KUKA KRL program: MyProgram_166().src

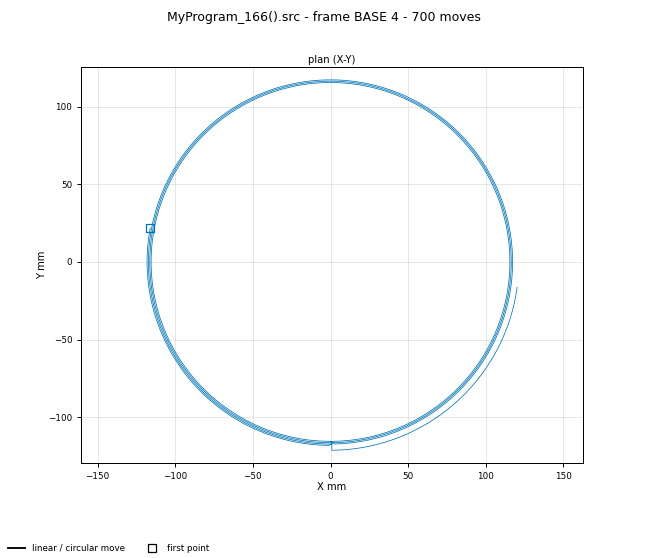
[picture p0: tool path of MyProgram_166().src in frame BASE 4, 700 of 700 moves have a stored position in this frame; points joined in program order, loops and branches not executed]
&ACCESS RVP
&REL 1
&PARAM TEMPLATE = C:\KRC\Roboter\Template\vorgabe
&PARAM EDITMASK = *
DEF MyProgram_166()
; ---- Setting reference (Base) ----
$BASE = BASE_DATA[4]

; --------------------------
; ---- Setting tool (TCP) ----
$TOOL = TOOL_DATA[3]
; --------------------------

$VEL.CP = VEL_APROX_PRINT
Startdeposition()
$VEL.CP = VEL_PRINT
LIN {X -116.0779,Y 21.7482,Z 125,A 166.5415,B 24.9441,C -1.7272,E1 24.8419,E2 279.4054} C_DIS
LIN {X -116.9015,Y 16.7566,Z 125,A 168.4487,B 24.9461,C -1.6962,E1 24.8412,E2 277.5607} C_DIS
LIN {X -117.4117,Y 12.7035,Z 125,A 170.2727,B 24.9469,C -1.6831,E1 24.8406,E2 275.757} C_DIS
LIN {X -117.7284,Y 9.3134,Z 125,A 171.8723,B 24.9474,C -1.6755,E1 24.8402,E2 274.1658} C_DIS
LIN {X -118.0302,Y 3.9618,Z 125,A 174.4618,B 24.948,C -1.6666,E1 24.8399,E2 271.5821} C_DIS
LIN {X -118.095,Y 0.6382,Z 125,A 176.1945,B 24.948,C -1.6663,E1 24.8398,E2 269.8396} C_DIS
LIN {X -118.0463,Y -3.4397,Z 125,A 178.1568,B 24.9484,C -1.6592,E1 24.8398,E2 267.8824} C_DIS
LIN {X -117.9024,Y -6.7675,Z 125,A 179.7767,B 24.9487,C -1.6541,E1 24.8401,E2 266.265} C_DIS
LIN {X -117.4382,Y -12.4501,Z 125,A -177.4787,B 24.9493,C -1.6442,E1 24.8408,E2 263.5274} C_DIS
LIN {X -117.0347,Y -15.812,Z 125,A -175.2833,B 24.9482,C -1.6622,E1 24.8416,E2 261.2762} C_DIS
LIN {X -116.456,Y -19.6147,Z 125,A -173.0042,B 24.9475,C -1.6738,E1 24.8427,E2 258.9558} C_DIS
LIN {X -115.3606,Y -25.2717,Z 125,A -171.1064,B 24.9504,C -1.627,E1 24.8438,E2 257.1584} C_DIS
LIN {X -113.6862,Y -31.9722,Z 125,A -167.6075,B 24.9507,C -1.6228,E1 24.8462,E2 253.6492} C_DIS
LIN {X -112.4267,Y -36.1525,Z 125,A -165.5854,B 24.9513,C -1.6123,E1 24.8479,E2 251.6404} C_DIS
LIN {X -111.457,Y -39.0393,Z 125,A -164.0611,B 24.9514,C -1.6098,E1 24.8493,E2 250.1133} C_DIS
LIN {X -110.0528,Y -42.8395,Z 125,A -162.0909,B 24.9518,C -1.6041,E1 24.8512,E2 248.1455} C_DIS
LIN {X -108.7242,Y -46.1068,Z 125,A -159.2633,B 24.9492,C -1.6468,E1 24.8545,E2 245.2007} C_DIS
LIN {X -105.8827,Y -52.303,Z 125,A -157.3666,B 24.9534,C -1.5771,E1 24.8566,E2 243.4597} C_DIS
LIN {X -103.1276,Y -57.545,Z 125,A -154.1935,B 24.9531,C -1.5818,E1 24.8608,E2 240.2585} C_DIS
LIN {X -101.6073,Y -60.1887,Z 125,A -152.6604,B 24.9532,C -1.5801,E1 24.8629,E2 238.7217} C_DIS
LIN {X -97.5843,Y -66.5143,Z 125,A -149.0981,B 24.954,C -1.5673,E1 24.8683,E2 235.1718} C_DIS
LIN {X -95.9307,Y -68.8777,Z 125,A -147.6463,B 24.954,C -1.566,E1 24.8706,E2 233.716} C_DIS
LIN {X -93.6134,Y -71.9949,Z 125,A -145.7524,B 24.9543,C -1.5617,E1 24.8738,E2 231.8231} C_DIS
LIN {X -91.4931,Y -74.6719,Z 125,A -144.0977,B 24.9545,C -1.5577,E1 24.8767,E2 230.1705} C_DIS
LIN {X -88.0813,Y -78.6665,Z 125,A -141.3029,B 24.9543,C -1.5623,E1 24.8819,E2 227.3518} C_DIS
LIN {X -85.8212,Y -81.1267,Z 125,A -139.7844,B 24.9547,C -1.5543,E1 24.8848,E2 225.8458} C_DIS
LIN {X -82.07,Y -84.9191,Z 125,A -137.0977,B 24.9548,C -1.553,E1 24.8901,E2 223.1508} C_DIS
LIN {X -78.6307,Y -88.1133,Z 125,A -134.9895,B 24.9555,C -1.5411,E1 24.8944,E2 221.0626} C_DIS
LIN {X -72.9131,Y -92.9008,Z 125,A -131.3391,B 24.9558,C -1.5355,E1 24.9023,E2 217.4116} C_DIS
LIN {X -68.4919,Y -96.206,Z 125,A -128.6806,B 24.9561,C -1.53,E1 24.9083,E2 214.7569} C_DIS
LIN {X -65.9216,Y -97.9856,Z 125,A -127.1661,B 24.9563,C -1.5274,E1 24.9117,E2 213.2434} C_DIS
LIN {X -62.3775,Y -100.2787,Z 125,A -125.0915,B 24.9564,C -1.5253,E1 24.9166,E2 211.167} C_DIS
LIN {X -58.5723,Y -102.548,Z 125,A -122.9855,B 24.9567,C -1.5203,E1 24.9217,E2 209.0667} C_DIS
LIN {X -55.7443,Y -104.1139,Z 125,A -120.7068,B 24.955,C -1.5497,E1 24.9275,E2 206.7118} C_DIS
LIN {X -51.6289,Y -106.2142,Z 125,A -119.1905,B 24.957,C -1.5146,E1 24.9311,E2 205.2748} C_DIS
LIN {X -48.5348,Y -107.6619,Z 125,A -117.4642,B 24.957,C -1.5158,E1 24.9355,E2 203.5415} C_DIS
LIN {X -42.3143,Y -110.2565,Z 125,A -114.3104,B 24.9574,C -1.5072,E1 24.9436,E2 200.401} C_DIS
LIN {X -39.7247,Y -111.2164,Z 125,A -112.6586,B 24.9567,C -1.5199,E1 24.948,E2 198.7157} C_DIS
LIN {X -35.4891,Y -112.6389,Z 125,A -110.3493,B 24.9565,C -1.5246,E1 24.9542,E2 196.3911} C_DIS
LIN {X -30.9043,Y -113.9809,Z 125,A -108.3462,B 24.9573,C -1.5089,E1 24.9595,E2 194.4221} C_DIS
LIN {X -27.7382,Y -114.7927,Z 125,A -106.8062,B 24.9575,C -1.5059,E1 24.9636,E2 192.8869} C_DIS
LIN {X -24.3093,Y -115.5686,Z 125,A -104.9791,B 24.9573,C -1.5106,E1 24.9687,E2 191.0466} C_DIS
LIN {X -20.8405,Y -116.2428,Z 125,A -103.3413,B 24.9575,C -1.5065,E1 24.9731,E2 189.4166} C_DIS
LIN {X -17.1768,Y -116.8418,Z 125,A -101.1085,B 24.9564,C -1.5257,E1 24.9794,E2 187.1365} C_DIS
LIN {X -13.728,Y -117.2956,Z 125,A -99.9123,B 24.9577,C -1.503,E1 24.9826,E2 185.9933} C_DIS
LIN {X -10.8458,Y -117.5971,Z 125,A -98.4243,B 24.9575,C -1.5066,E1 24.9868,E2 184.4959} C_DIS
LIN {X -7.1405,Y -117.8818,Z 125,A -96.3974,B 24.9569,C -1.5168,E1 24.9925,E2 182.444} C_DIS
LIN {X -1.2408,Y -118.0908,Z 125,A -93.9033,B 24.9578,C -1.5003,E1 24.9993,E2 179.9888} C_DIS
LIN {X -1.2408,Y -118.0908,Z 125,A -93.9033,B 24.9578,C -1.5003,E1 24.9993,E2 179.9888} C_DIS
Enddeposition()
LIN {X 0.8351,Y -117.2293,Z 125,A -92.7873,B 24.9567,C -1.5205,E1 25.0026,E2 178.825} C_DIS
Startdeposition()
$VEL.CP = VEL_PRINT
LIN {X -1.6148,Y -117.2225,Z 125,A -94.8526,B 24.9589,C -1.4811,E1 24.9966,E2 180.9837} C_DIS
LIN {X -6.2337,Y -117.0668,Z 125,A -96.9986,B 24.9586,C -1.4859,E1 24.9906,E2 183.1186} C_DIS
LIN {X -9.7696,Y -116.8254,Z 125,A -98.7217,B 24.9586,C -1.4863,E1 24.9858,E2 184.8415} C_DIS
LIN {X -13.4236,Y -116.4615,Z 125,A -100.2293,B 24.9579,C -1.4993,E1 24.9817,E2 186.3191} C_DIS
LIN {X -17.0983,Y -115.9804,Z 125,A -102.4267,B 24.9588,C -1.4825,E1 24.9755,E2 188.5581} C_DIS
LIN {X -20.6841,Y -115.3933,Z 125,A -104.0258,B 24.9584,C -1.4909,E1 24.9712,E2 190.1388} C_DIS
LIN {X -23.7178,Y -114.8082,Z 125,A -105.6383,B 24.9586,C -1.487,E1 24.9667,E2 191.7624} C_DIS
LIN {X -27.5658,Y -113.9457,Z 125,A -107.5616,B 24.9586,C -1.4882,E1 24.9615,E2 193.6855} C_DIS
LIN {X -31.5414,Y -112.9104,Z 125,A -109.9728,B 24.9594,C -1.4718,E1 24.9549,E2 196.1393} C_DIS
LIN {X -34.9646,Y -111.8972,Z 125,A -111.6053,B 24.9591,C -1.478,E1 24.9505,E2 197.7599} C_DIS
LIN {X -39.9943,Y -110.1995,Z 125,A -113.8892,B 24.9582,C -1.4937,E1 24.9446,E2 200.0108} C_DIS
LIN {X -42.7939,Y -109.1427,Z 125,A -115.7888,B 24.9592,C -1.4762,E1 24.9396,E2 201.9561} C_DIS
LIN {X -46.2472,Y -107.7268,Z 125,A -117.2748,B 24.9583,C -1.4927,E1 24.9358,E2 203.4063} C_DIS
LIN {X -49.5329,Y -106.2541,Z 125,A -118.8769,B 24.9578,C -1.5016,E1 24.9318,E2 204.9913} C_DIS
LIN {X -54.7369,Y -103.6693,Z 125,A -121.9132,B 24.958,C -1.4967,E1 24.9242,E2 208.0474} C_DIS
LIN {X -59.799,Y -100.8343,Z 125,A -124.7248,B 24.9577,C -1.5018,E1 24.9174,E2 210.8553} C_DIS
LIN {X -63.9365,Y -98.2653,Z 125,A -127.107,B 24.9575,C -1.5053,E1 24.9118,E2 213.2365} C_DIS
LIN {X -67.376,Y -95.9386,Z 125,A -129.3507,B 24.9579,C -1.4996,E1 24.9066,E2 215.5015} C_DIS
LIN {X -71.4168,Y -92.9683,Z 125,A -131.5025,B 24.9569,C -1.5167,E1 24.9018,E2 217.6203} C_DIS
LIN {X -73.3854,Y -91.4238,Z 125,A -133.2937,B 24.9581,C -1.4949,E1 24.8978,E2 219.47} C_DIS
LIN {X -76.5724,Y -88.7728,Z 125,A -134.9135,B 24.9569,C -1.516,E1 24.8945,E2 221.0461} C_DIS
LIN {X -79.2536,Y -86.3846,Z 125,A -136.6869,B 24.9568,C -1.5188,E1 24.8908,E2 222.8199} C_DIS
LIN {X -81.8829,Y -83.8994,Z 125,A -138.5802,B 24.9568,C -1.5172,E1 24.887,E2 224.7249} C_DIS
LIN {X -85.2057,Y -80.5202,Z 125,A -140.8343,B 24.9564,C -1.5249,E1 24.8826,E2 226.9703} C_DIS
LIN {X -88.1501,Y -77.2854,Z 125,A -142.9732,B 24.9562,C -1.5297,E1 24.8786,E2 229.1073} C_DIS
LIN {X -91.033,Y -73.8677,Z 125,A -144.9562,B 24.9554,C -1.5434,E1 24.8751,E2 231.0669} C_DIS
LIN {X -93.5183,Y -70.6958,Z 125,A -146.9961,B 24.9553,C -1.5452,E1 24.8716,E2 233.1121} C_DIS
LIN {X -95.4795,Y -68.0229,Z 125,A -148.6269,B 24.9551,C -1.5489,E1 24.869,E2 234.7422} C_DIS
LIN {X -97.7454,Y -64.7249,Z 125,A -151.0294,B 24.9558,C -1.5354,E1 24.8652,E2 237.1887} C_DIS
LIN {X -99.8083,Y -61.5001,Z 125,A -152.5944,B 24.9548,C -1.553,E1 24.8629,E2 238.7199} C_DIS
LIN {X -102.0444,Y -57.7129,Z 125,A -154.8515,B 24.9548,C -1.5544,E1 24.8598,E2 240.9854} C_DIS
LIN {X -104.1752,Y -53.7698,Z 125,A -156.8916,B 24.954,C -1.5667,E1 24.8571,E2 243.0071} C_DIS
LIN {X -106.0255,Y -50.024,Z 125,A -159.5909,B 24.9552,C -1.5456,E1 24.8538,E2 245.7713} C_DIS
LIN {X -107.9815,Y -45.6448,Z 125,A -161.2325,B 24.9532,C -1.5811,E1 24.8521,E2 247.3372} C_DIS
LIN {X -109.202,Y -42.6428,Z 125,A -162.8678,B 24.953,C -1.5837,E1 24.8504,E2 248.9757} C_DIS
LIN {X -110.5039,Y -39.1465,Z 125,A -164.7261,B 24.9528,C -1.5877,E1 24.8486,E2 250.8349} C_DIS
LIN {X -111.655,Y -35.7315,Z 125,A -166.5622,B 24.9526,C -1.5899,E1 24.847,E2 252.676} C_DIS
LIN {X -112.8242,Y -31.8458,Z 125,A -169.1513,B 24.9537,C -1.5714,E1 24.845,E2 255.3243} C_DIS
LIN {X -114.074,Y -27.037,Z 125,A -170.9059,B 24.9517,C -1.6063,E1 24.8439,E2 257.006} C_DIS
LIN {X -115.1522,Y -21.9871,Z 125,A -173.4355,B 24.9512,C -1.614,E1 24.8424,E2 259.5321} C_DIS
LIN {X -116.2866,Y -14.8631,Z 125,A -176.9173,B 24.9504,C -1.627,E1 24.841,E2 263.0037} C_DIS
LIN {X -116.6475,Y -11.7067,Z 125,A -178.8834,B 24.9511,C -1.6152,E1 24.8404,E2 265.0097} C_DIS
LIN {X -116.9276,Y -8.4665,Z 125,A 179.86,B 24.95,C -1.6339,E1 24.8401,E2 266.2295} C_DIS
LIN {X -117.1256,Y -5.0025,Z 125,A 178.1548,B 24.9497,C -1.639,E1 24.8399,E2 267.9326} C_DIS
LIN {X -117.2264,Y -1.3455,Z 125,A 176.2701,B 24.9495,C -1.6409,E1 24.8398,E2 269.8242} C_DIS
LIN {X -117.2105,Y 2.2703,Z 125,A 174.6527,B 24.9488,C -1.6527,E1 24.8398,E2 271.423} C_DIS
LIN {X -117.0681,Y 6.2092,Z 125,A 172.3947,B 24.9493,C -1.6456,E1 24.8401,E2 273.7118} C_DIS
LIN {X -116.7635,Y 10.4787,Z 125,A 170.5424,B 24.9482,C -1.6621,E1 24.8405,E2 275.5357} C_DIS
LIN {X -116.1042,Y 16.2268,Z 125,A 167.5686,B 24.948,C -1.6654,E1 24.8415,E2 278.5195} C_DIS
LIN {X -115.4155,Y 20.5602,Z 125,A 165.5301,B 24.9473,C -1.6767,E1 24.8425,E2 280.5433} C_DIS
LIN {X -114.1275,Y 26.8053,Z 125,A 162.2668,B 24.9471,C -1.6808,E1 24.8444,E2 283.816} C_DIS
LIN {X -112.9284,Y 31.478,Z 125,A 159.9483,B 24.9465,C -1.6899,E1 24.846,E2 286.1263} C_DIS
LIN {X -112.0005,Y 34.6314,Z 125,A 158.3319,B 24.9462,C -1.6946,E1 24.8474,E2 287.7407} C_DIS
LIN {X -110.8147,Y 38.2607,Z 125,A 156.4862,B 24.9458,C -1.7013,E1 24.849,E2 289.581} C_DIS
LIN {X -108.853,Y 43.5312,Z 125,A 153.6729,B 24.9454,C -1.7072,E1 24.8518,E2 292.396} C_DIS
LIN {X -107.4588,Y 46.8619,Z 125,A 151.9605,B 24.9449,C -1.7148,E1 24.8537,E2 294.0998} C_DIS
LIN {X -105.8573,Y 50.3772,Z 125,A 150.0068,B 24.9447,C -1.7179,E1 24.856,E2 296.0569} C_DIS
LIN {X -104.1375,Y 53.8435,Z 125,A 147.8473,B 24.945,C -1.7126,E1 24.8587,E2 298.2405} C_DIS
LIN {X -101.4971,Y 58.6675,Z 125,A 144.7651,B 24.9455,C -1.7046,E1 24.863,E2 301.3579} C_DIS
LIN {X -98.9869,Y 62.8124,Z 125,A 143.1773,B 24.9431,C -1.7431,E1 24.8653,E2 302.8621} C_DIS
LIN {X -95.8292,Y 67.5327,Z 125,A 139.7815,B 24.9442,C -1.7255,E1 24.8707,E2 306.3166} C_DIS
LIN {X -93.5753,Y 70.6199,Z 125,A 138.8928,B 24.9412,C -1.7708,E1 24.872,E2 307.1016} C_DIS
LIN {X -91.6258,Y 73.1332,Z 125,A 136.9431,B 24.942,C -1.7586,E1 24.8754,E2 309.0896} C_DIS
LIN {X -89.5071,Y 75.7106,Z 125,A 135.1595,B 24.9422,C -1.7566,E1 24.8786,E2 310.8862} C_DIS
LIN {X -87.2439,Y 78.3068,Z 125,A 133.6175,B 24.9415,C -1.7668,E1 24.8814,E2 312.4109} C_DIS
LIN {X -84.5415,Y 81.2171,Z 125,A 131.5821,B 24.9415,C -1.7678,E1 24.8853,E2 314.4529} C_DIS
LIN {X -81.1171,Y 84.6378,Z 125,A 129.058,B 24.9415,C -1.7669,E1 24.8904,E2 316.9895} C_DIS
LIN {X -77.8834,Y 87.623,Z 125,A 126.6566,B 24.9418,C -1.7616,E1 24.8954,E2 319.4132} C_DIS
LIN {X -75.3603,Y 89.803,Z 125,A 125.2726,B 24.9409,C -1.7754,E1 24.8983,E2 320.7697} C_DIS
LIN {X -72.6864,Y 91.979,Z 125,A 123.3436,B 24.9413,C -1.769,E1 24.9026,E2 322.721} C_DIS
LIN {X -70.1029,Y 93.9637,Z 125,A 121.5268,B 24.9417,C -1.7631,E1 24.9067,E2 324.5585} C_DIS
LIN {X -66.7194,Y 96.3951,Z 125,A 119.9213,B 24.9403,C -1.7851,E1 24.9103,E2 326.1172} C_DIS
LIN {X -64.0955,Y 98.1604,Z 125,A 118.303,B 24.9403,C -1.7851,E1 24.9141,E2 327.7408} C_DIS
LIN {X -61.2043,Y 99.988,Z 125,A 116.6727,B 24.94,C -1.7899,E1 24.9179,E2 329.3646} C_DIS
LIN {X -57.3374,Y 102.2541,Z 125,A 114.5912,B 24.9394,C -1.7984,E1 24.9229,E2 331.432} C_DIS
LIN {X -54.0312,Y 104.0408,Z 125,A 112.8232,B 24.939,C -1.8044,E1 24.9272,E2 333.1908} C_DIS
LIN {X -48.6263,Y 106.6732,Z 125,A 109.7819,B 24.939,C -1.8047,E1 24.9349,E2 336.2391} C_DIS
LIN {X -45.4531,Y 108.0623,Z 125,A 108.1017,B 24.9387,C -1.8078,E1 24.9392,E2 337.916} C_DIS
LIN {X -39.0031,Y 110.5542,Z 125,A 104.7495,B 24.9384,C -1.8134,E1 24.948,E2 341.2617} C_DIS
LIN {X -35.6874,Y 111.6693,Z 125,A 102.4145,B 24.94,C -1.7889,E1 24.9543,E2 343.6592} C_DIS
LIN {X -31.5151,Y 112.9171,Z 125,A 100.777,B 24.9385,C -1.812,E1 24.9586,E2 345.2443} C_DIS
LIN {X -23.9618,Y 114.7581,Z 125,A 97.0607,B 24.938,C -1.8192,E1 24.9687,E2 348.9488} C_DIS
LIN {X -20.7726,Y 115.3774,Z 125,A 95.4352,B 24.938,C -1.8188,E1 24.9731,E2 350.5768} C_DIS
LIN {X -16.7737,Y 116.0265,Z 125,A 93.482,B 24.9378,C -1.8213,E1 24.9785,E2 352.5258} C_DIS
LIN {X -13.0492,Y 116.5054,Z 125,A 91.5989,B 24.9378,C -1.8203,E1 24.9837,E2 354.4126} C_DIS
LIN {X -9.6564,Y 116.8344,Z 125,A 89.9798,B 24.9377,C -1.8232,E1 24.9882,E2 356.0256} C_DIS
LIN {X -6.466,Y 117.0539,Z 125,A 88.4343,B 24.9377,C -1.8245,E1 24.9925,E2 357.5684} C_DIS
LIN {X -2.5675,Y 117.205,Z 125,A 86.4811,B 24.9377,C -1.8231,E1 24.998,E2 359.5254} C_DIS
LIN {X 0.8052,Y 117.2297,Z 125,A 84.8525,B 24.9377,C -1.8243,E1 25.0025,E2 361.1511} C_DIS
LIN {X 4.8542,Y 117.132,Z 125,A 82.9127,B 24.9375,C -1.8262,E1 25.0079,E2 363.0858} C_DIS
LIN {X 8.3744,Y 116.9338,Z 125,A 81.1059,B 24.9377,C -1.8225,E1 25.013,E2 364.9007} C_DIS
LIN {X 11.9675,Y 116.6202,Z 125,A 79.4204,B 24.9375,C -1.8257,E1 25.0176,E2 366.5776} C_DIS
LIN {X 15.1732,Y 116.2464,Z 125,A 77.8138,B 24.9376,C -1.8241,E1 25.0221,E2 368.1868} C_DIS
LIN {X 18.973,Y 115.6875,Z 125,A 75.8997,B 24.9378,C -1.8219,E1 25.0274,E2 370.1043} C_DIS
LIN {X 22.6611,Y 115.0224,Z 125,A 74.0299,B 24.938,C -1.8194,E1 25.0325,E2 371.9778} C_DIS
LIN {X 26.259,Y 114.2537,Z 125,A 72.3871,B 24.9375,C -1.8254,E1 25.037,E2 373.6042} C_DIS
LIN {X 31.9221,Y 112.8025,Z 125,A 69.1138,B 24.9389,C -1.805,E1 25.0459,E2 376.9205} C_DIS
LIN {X 35.1622,Y 111.8359,Z 125,A 67.7111,B 24.9383,C -1.8149,E1 25.0496,E2 378.2975} C_DIS
LIN {X 39.4824,Y 110.386,Z 125,A 65.1137,B 24.9395,C -1.7963,E1 25.0565,E2 380.9335} C_DIS
LIN {X 43.0096,Y 109.0579,Z 125,A 63.7611,B 24.9382,C -1.8165,E1 25.0599,E2 382.2355} C_DIS
LIN {X 46.5591,Y 107.5908,Z 125,A 62.1231,B 24.9376,C -1.8252,E1 25.0641,E2 383.8489} C_DIS
LIN {X 50.5222,Y 105.7876,Z 125,A 59.5155,B 24.9392,C -1.801,E1 25.0708,E2 386.5072} C_DIS
LIN {X 55.0343,Y 103.5126,Z 125,A 57.2937,B 24.9387,C -1.8089,E1 25.0763,E2 388.704} C_DIS
LIN {X 58.1162,Y 101.8138,Z 125,A 55.5703,B 24.9388,C -1.8063,E1 25.0805,E2 390.4285} C_DIS
LIN {X 61.5238,Y 99.7934,Z 125,A 53.5557,B 24.9393,C -1.7998,E1 25.0853,E2 392.4523} C_DIS
LIN {X 64.3245,Y 98.0095,Z 125,A 51.3769,B 24.9412,C -1.7719,E1 25.0905,E2 394.6897} C_DIS
LIN {X 68.1982,Y 95.3544,Z 125,A 49.7395,B 24.9394,C -1.798,E1 25.0941,E2 396.26} C_DIS
LIN {X 73.4759,Y 91.3505,Z 125,A 46.4859,B 24.9399,C -1.7913,E1 25.1013,E2 399.5175} C_DIS
LIN {X 76.1243,Y 89.1546,Z 125,A 44.995,B 24.9395,C -1.7968,E1 25.1045,E2 400.9895} C_DIS
LIN {X 78.7411,Y 86.8548,Z 125,A 43.1919,B 24.94,C -1.7887,E1 25.1082,E2 402.8046} C_DIS
LIN {X 81.3986,Y 84.3665,Z 125,A 41.3875,B 24.9404,C -1.7838,E1 25.1119,E2 404.6131} C_DIS
LIN {X 84.8199,Y 80.9275,Z 125,A 39.072,B 24.9405,C -1.7812,E1 25.1164,E2 406.9249} C_DIS
LIN {X 87.4068,Y 78.1248,Z 125,A 37.2011,B 24.9408,C -1.7766,E1 25.12,E2 408.7982} C_DIS
LIN {X 89.8127,Y 75.3486,Z 125,A 35.5173,B 24.9408,C -1.7776,E1 25.123,E2 410.4721} C_DIS
LIN {X 93.0756,Y 71.2775,Z 125,A 32.7485,B 24.9419,C -1.7612,E1 25.1279,E2 413.2667} C_DIS
LIN {X 97.1409,Y 65.6284,Z 125,A 29.4447,B 24.9421,C -1.7571,E1 25.1332,E2 416.5641} C_DIS
LIN {X 99.395,Y 62.1617,Z 125,A 27.5293,B 24.9421,C -1.7567,E1 25.136,E2 418.4708} C_DIS
LIN {X 100.6871,Y 60.0479,Z 125,A 25.6319,B 24.9445,C -1.7213,E1 25.1389,E2 420.442} C_DIS
LIN {X 102.9107,Y 56.1507,Z 125,A 24.0908,B 24.9429,C -1.7458,E1 25.1409,E2 421.9173} C_DIS
LIN {X 104.2182,Y 53.6856,Z 125,A 22.891,B 24.9426,C -1.7497,E1 25.1424,E2 423.1015} C_DIS
LIN {X 105.5158,Y 51.0879,Z 125,A 21.253,B 24.9436,C -1.7353,E1 25.1444,E2 424.7647} C_DIS
LIN {X 106.9734,Y 47.9601,Z 125,A 19.6193,B 24.9437,C -1.733,E1 25.1463,E2 426.3951} C_DIS
LIN {X 108.5068,Y 44.3819,Z 125,A 17.8754,B 24.9436,C -1.7349,E1 25.1482,E2 428.1248} C_DIS
LIN {X 109.8782,Y 40.8741,Z 125,A 15.821,B 24.9446,C -1.7193,E1 25.1503,E2 430.2046} C_DIS
LIN {X 110.8838,Y 38.0607,Z 125,A 13.7234,B 24.9468,C -1.6848,E1 25.1523,E2 432.3716} C_DIS
LIN {X 112.3926,Y 33.3367,Z 125,A 11.4302,B 24.9468,C -1.6835,E1 25.154,E2 434.6548} C_DIS
LIN {X 113.5969,Y 28.9696,Z 125,A 9.8432,B 24.9454,C -1.7063,E1 25.1551,E2 436.179} C_DIS
LIN {X 114.5094,Y 25.1205,Z 125,A 7.9293,B 24.9458,C -1.7012,E1 25.1563,E2 438.0939} C_DIS
LIN {X 115.254,Y 21.4586,Z 125,A 5.9882,B 24.9465,C -1.6899,E1 25.1574,E2 440.0503} C_DIS
LIN {X 115.8309,Y 18.074,Z 125,A 4.4194,B 24.9465,C -1.6898,E1 25.1581,E2 441.6101} C_DIS
LIN {X 116.3583,Y 14.3051,Z 125,A 2.5225,B 24.947,C -1.682,E1 25.1588,E2 443.5142} C_DIS
LIN {X 116.7249,Y 10.8971,Z 125,A 0.9515,B 24.947,C -1.6816,E1 25.1592,E2 445.0768} C_DIS
LIN {X 116.9915,Y 7.5207,Z 125,A -0.808,B 24.9477,C -1.6712,E1 25.1595,E2 446.8502} C_DIS
LIN {X 117.1775,Y 3.5875,Z 125,A -2.6481,B 24.9477,C -1.669,E1 25.1597,E2 448.6846} C_DIS
LIN {X 117.2324,Y -0.4409,Z 125,A -4.6079,B 24.9482,C -1.663,E1 25.1597,E2 450.6469} C_DIS
LIN {X 117.1621,Y -4.0889,Z 125,A -6.2539,B 24.9482,C -1.6637,E1 25.1597,E2 452.2814} C_DIS
LIN {X 117.0279,Y -6.9364,Z 125,A -7.8163,B 24.9489,C -1.6511,E1 25.1594,E2 453.8644} C_DIS
LIN {X 116.7319,Y -10.821,Z 125,A -9.6054,B 24.9489,C -1.6504,E1 25.159,E2 455.6445} C_DIS
LIN {X 116.3079,Y -14.6987,Z 125,A -11.5635,B 24.9495,C -1.6416,E1 25.1584,E2 457.6116} C_DIS
LIN {X 115.7525,Y -18.5812,Z 125,A -13.4711,B 24.9499,C -1.6358,E1 25.1576,E2 459.5217} C_DIS
LIN {X 115.0246,Y -22.6497,Z 125,A -15.5647,B 24.9505,C -1.6257,E1 25.1565,E2 461.6268} C_DIS
LIN {X 114.0065,Y -27.3162,Z 125,A -17.5785,B 24.95,C -1.6335,E1 25.1553,E2 463.6106} C_DIS
LIN {X 112.2087,Y -33.9568,Z 125,A -21.0165,B 24.9509,C -1.619,E1 25.1527,E2 467.063} C_DIS
LIN {X 110.3917,Y -39.4659,Z 125,A -23.9646,B 24.9518,C -1.6046,E1 25.1501,E2 470.0284} C_DIS
LIN {X 109.0827,Y -42.9465,Z 125,A -25.693,B 24.9518,C -1.6032,E1 25.1483,E2 471.7506} C_DIS
LIN {X 107.9815,Y -45.6448,Z 125,A -27.637,B 24.9536,C -1.5741,E1 25.1462,E2 473.7525} C_DIS
LIN {X 106.33,Y -49.3697,Z 125,A -29.6176,B 24.9539,C -1.5685,E1 25.1438,E2 475.7356} C_DIS
LIN {X 104.5358,Y -53.0641,Z 125,A -30.9535,B 24.9524,C -1.5944,E1 25.1423,E2 477.0034} C_DIS
LIN {X 101.108,Y -59.3358,Z 125,A -34.5861,B 24.9534,C -1.5773,E1 25.1373,E2 480.6573} C_DIS
LIN {X 98.6083,Y -63.4023,Z 125,A -36.856,B 24.9536,C -1.5736,E1 25.1339,E2 482.9245} C_DIS
LIN {X 94.9914,Y -68.7062,Z 125,A -39.9233,B 24.9539,C -1.568,E1 25.1291,E2 485.9899} C_DIS
LIN {X 92.367,Y -72.1953,Z 125,A -42.2211,B 24.9547,C -1.5544,E1 25.1252,E2 488.3089} C_DIS
LIN {X 89.4516,Y -75.7757,Z 125,A -44.5234,B 24.9552,C -1.5462,E1 25.121,E2 490.6199} C_DIS
LIN {X 85.9649,Y -79.7104,Z 125,A -47.0053,B 24.9554,C -1.5437,E1 25.1164,E2 493.0966} C_DIS
LIN {X 82.9275,Y -82.8668,Z 125,A -49.6064,B 24.9569,C -1.5168,E1 25.1112,E2 495.7502} C_DIS
LIN {X 79.9206,Y -85.769,Z 125,A -51.0702,B 24.9556,C -1.539,E1 25.1083,E2 497.1555} C_DIS
LIN {X 77.0081,Y -88.3924,Z 125,A -53.0042,B 24.9559,C -1.5337,E1 25.1043,E2 499.0944} C_DIS
LIN {X 73.7199,Y -91.1528,Z 125,A -55.9662,B 24.9585,C -1.4888,E1 25.0977,E2 502.1512} C_DIS
LIN {X 69.1598,Y -94.6593,Z 125,A -58.4359,B 24.9579,C -1.4986,E1 25.0922,E2 504.589} C_DIS
LIN {X 65.6786,Y -97.1069,Z 125,A -59.9349,B 24.9566,C -1.5214,E1 25.0889,E2 506.0291} C_DIS
LIN {X 62.4525,Y -99.2133,Z 125,A -61.9006,B 24.9571,C -1.5138,E1 25.0842,E2 508.0063} C_DIS
LIN {X 58.2312,Y -101.7477,Z 125,A -64.8395,B 24.9587,C -1.4848,E1 25.077,E2 511.0049} C_DIS
LIN {X 54.2238,Y -103.9395,Z 125,A -66.4275,B 24.9572,C -1.5106,E1 25.0732,E2 512.5273} C_DIS
LIN {X 51.658,Y -105.2383,Z 125,A -68.2403,B 24.9584,C -1.4895,E1 25.0686,E2 514.3852} C_DIS
LIN {X 48.4985,Y -106.7308,Z 125,A -69.5497,B 24.9576,C -1.5051,E1 25.0654,E2 515.6542} C_DIS
LIN {X 45.4161,Y -108.0779,Z 125,A -71.2077,B 24.9577,C -1.502,E1 25.0611,E2 517.3157} C_DIS
LIN {X 41.49,Y -109.645,Z 125,A -73.4705,B 24.9584,C -1.4901,E1 25.0551,E2 519.6017} C_DIS
LIN {X 38.4727,Y -110.7403,Z 125,A -75.1612,B 24.9588,C -1.4825,E1 25.0507,E2 521.3071} C_DIS
LIN {X 35.2715,Y -111.802,Z 125,A -76.5266,B 24.9582,C -1.4934,E1 25.0471,E2 522.6441} C_DIS
LIN {X 31.869,Y -112.8176,Z 125,A -78.1994,B 24.9582,C -1.4943,E1 25.0426,E2 524.3119} C_DIS
LIN {X 27.2402,Y -114.0251,Z 125,A -80.6192,B 24.9585,C -1.4882,E1 25.036,E2 526.7426} C_DIS
LIN {X 23.6964,Y -114.8126,Z 125,A -82.2846,B 24.9583,C -1.4915,E1 25.0315,E2 528.3979} C_DIS
LIN {X 20.0067,Y -115.5146,Z 125,A -84.1756,B 24.9585,C -1.4875,E1 25.0263,E2 530.2964} C_DIS
LIN {X 16.5297,Y -116.0612,Z 125,A -85.818,B 24.9585,C -1.4898,E1 25.0218,E2 531.9318} C_DIS
LIN {X 13.056,Y -116.5046,Z 125,A -87.6066,B 24.9587,C -1.4852,E1 25.0168,E2 533.7298} C_DIS
LIN {X 9.5655,Y -116.8417,Z 125,A -89.2068,B 24.9584,C -1.4895,E1 25.0124,E2 535.319} C_DIS
LIN {X 6.4115,Y -117.057,Z 125,A -90.8279,B 24.9587,C -1.4854,E1 25.0078,E2 536.9492} C_DIS
LIN {X 2.6212,Y -117.204,Z 125,A -92.7006,B 24.9587,C -1.4839,E1 25.0026,E2 538.825} C_DIS
LIN {X 2.6212,Y -117.204,Z 125,A -92.7006,B 24.9587,C -1.4839,E1 25.0026,E2 538.825} C_DIS
Enddeposition()
LIN {X 0.8327,Y -116.3647,Z 125,A -93.4098,B 24.9575,C -1.5063,E1 25.0008,E2 539.4811} C_DIS
Startdeposition()
$VEL.CP = VEL_PRINT
LIN {X 4.9481,Y -116.2633,Z 125,A -90.7671,B 24.9559,C -1.5346,E1 25.0083,E2 536.7719} C_DIS
LIN {X 7.905,Y -116.0998,Z 125,A -89.3433,B 24.9559,C -1.5337,E1 25.0123,E2 535.3509} C_DIS
LIN {X 11.4063,Y -115.8104,Z 125,A -87.4778,B 24.9555,C -1.5407,E1 25.0175,E2 533.4698} C_DIS
LIN {X 15.2906,Y -115.3601,Z 125,A -85.6407,B 24.9557,C -1.5379,E1 25.0226,E2 531.6406} C_DIS
LIN {X 19.057,Y -114.7976,Z 125,A -83.811,B 24.9557,C -1.5373,E1 25.0276,E2 529.8143} C_DIS
LIN {X 22.4288,Y -114.1875,Z 125,A -82.0603,B 24.9555,C -1.5416,E1 25.0324,E2 528.0555} C_DIS
LIN {X 26.3488,Y -113.3464,Z 125,A -80.1614,B 24.9555,C -1.54,E1 25.0376,E2 526.1628} C_DIS
LIN {X 33.1245,Y -111.5545,Z 125,A -77.0897,B 24.9564,C -1.5262,E1 25.0458,E2 523.1286} C_DIS
LIN {X 38.2794,Y -109.8927,Z 125,A -74.1715,B 24.9555,C -1.541,E1 25.0536,E2 520.1809} C_DIS
LIN {X 43.0824,Y -108.1012,Z 125,A -71.6154,B 24.9552,C -1.5459,E1 25.0603,E2 517.6188} C_DIS
LIN {X 45.8898,Y -106.9402,Z 125,A -69.9262,B 24.9546,C -1.5571,E1 25.0647,E2 515.9071} C_DIS
LIN {X 49.356,Y -105.3836,Z 125,A -67.8384,B 24.9538,C -1.5702,E1 25.0701,E2 513.7935} C_DIS
LIN {X 52.3322,Y -103.9397,Z 125,A -66.4157,B 24.9542,C -1.5632,E1 25.0736,E2 512.3911} C_DIS
LIN {X 55.551,Y -102.2533,Z 125,A -64.7028,B 24.9542,C -1.5628,E1 25.0778,E2 510.6841} C_DIS
LIN {X 60.8645,Y -99.1837,Z 125,A -61.6901,B 24.9539,C -1.568,E1 25.085,E2 507.6684} C_DIS
LIN {X 64.0066,Y -97.1844,Z 125,A -59.9135,B 24.9539,C -1.5689,E1 25.0892,E2 505.8954} C_DIS
LIN {X 67.4736,Y -94.8102,Z 125,A -57.8425,B 24.9536,C -1.5733,E1 25.0939,E2 503.8212} C_DIS
LIN {X 70.3783,Y -92.6763,Z 125,A -55.679,B 24.9523,C -1.5955,E1 25.0989,E2 501.6131} C_DIS
LIN {X 73.1329,Y -90.5166,Z 125,A -54.3763,B 24.9533,C -1.5794,E1 25.1016,E2 500.3533} C_DIS
LIN {X 75.8784,Y -88.2293,Z 125,A -52.4857,B 24.9527,C -1.5896,E1 25.1057,E2 498.4459} C_DIS
LIN {X 78.3863,Y -86.008,Z 125,A -50.1834,B 24.9505,C -1.6247,E1 25.1106,E2 496.0702} C_DIS
LIN {X 82.3017,Y -82.2712,Z 125,A -48.4093,B 24.9527,C -1.5886,E1 25.1139,E2 494.3886} C_DIS
LIN {X 84.9762,Y -79.5033,Z 125,A -46.4754,B 24.9523,C -1.5953,E1 25.1176,E2 492.4474} C_DIS
LIN {X 87.022,Y -77.2596,Z 125,A -44.1386,B 24.9496,C -1.6395,E1 25.1221,E2 490.0168} C_DIS
LIN {X 90.5219,Y -73.1264,Z 125,A -42.2579,B 24.9515,C -1.6088,E1 25.1253,E2 488.217} C_DIS
LIN {X 93.2711,Y -69.5866,Z 125,A -40.1952,B 24.9515,C -1.608,E1 25.1288,E2 486.1661} C_DIS
LIN {X 94.966,Y -67.2552,Z 125,A -38.7658,B 24.9513,C -1.6124,E1 25.1311,E2 484.7332} C_DIS
LIN {X 97.2738,Y -63.871,Z 125,A -36.7352,B 24.9509,C -1.6188,E1 25.1343,E2 482.6977} C_DIS
LIN {X 99.3505,Y -60.59,Z 125,A -34.7667,B 24.9504,C -1.627,E1 25.1372,E2 480.7196} C_DIS
LIN {X 101.8737,Y -56.2469,Z 125,A -32.4456,B 24.9504,C -1.627,E1 25.1404,E2 478.4107} C_DIS
LIN {X 103.0292,Y -54.0984,Z 125,A -31.194,B 24.95,C -1.6331,E1 25.1421,E2 477.1514} C_DIS
LIN {X 104.4321,Y -51.3392,Z 125,A -29.5571,B 24.9494,C -1.6431,E1 25.1441,E2 475.4997} C_DIS
LIN {X 107.1632,Y -45.3621,Z 125,A -26.72,B 24.95,C -1.6339,E1 25.1473,E2 472.6996} C_DIS
LIN {X 108.6215,Y -41.7535,Z 125,A -24.4268,B 24.9485,C -1.6579,E1 25.1497,E2 470.3625} C_DIS
LIN {X 109.9608,Y -38.0854,Z 125,A -22.328,B 24.9476,C -1.6725,E1 25.1517,E2 468.2411} C_DIS
LIN {X 111.2355,Y -34.1816,Z 125,A -20.5996,B 24.9481,C -1.6647,E1 25.1531,E2 466.5407} C_DIS
LIN {X 112.3561,Y -30.2945,Z 125,A -18.356,B 24.9469,C -1.6833,E1 25.1548,E2 464.2663} C_DIS
LIN {X 113.3322,Y -26.4105,Z 125,A -16.0227,B 24.9454,C -1.7072,E1 25.1564,E2 461.8903} C_DIS
LIN {X 114.2894,Y -21.8995,Z 125,A -14.4512,B 24.9471,C -1.6807,E1 25.1572,E2 460.3903} C_DIS
LIN {X 114.9123,Y -18.3615,Z 125,A -12.5629,B 24.9463,C -1.6922,E1 25.158,E2 458.486} C_DIS
LIN {X 115.4121,Y -14.8894,Z 125,A -10.9219,B 24.9463,C -1.6937,E1 25.1586,E2 456.8512} C_DIS
LIN {X 115.7732,Y -11.7618,Z 125,A -9.3217,B 24.9458,C -1.7012,E1 25.1591,E2 455.2428} C_DIS
LIN {X 116.1008,Y -7.8896,Z 125,A -7.4965,B 24.9456,C -1.7032,E1 25.1595,E2 453.4236} C_DIS
LIN {X 116.263,Y -4.9552,Z 125,A -6.0967,B 24.9455,C -1.7057,E1 25.1597,E2 452.0263} C_DIS
LIN {X 116.3627,Y -1.3165,Z 125,A -4.2057,B 24.9448,C -1.7162,E1 25.1597,E2 450.1216} C_DIS
LIN {X 116.3463,Y 2.2807,Z 125,A -2.5259,B 24.9448,C -1.7177,E1 25.1597,E2 448.4485} C_DIS
LIN {X 116.2044,Y 6.1835,Z 125,A -0.534,B 24.9441,C -1.7272,E1 25.1595,E2 446.4459} C_DIS
LIN {X 115.9788,Y 9.5194,Z 125,A 0.997,B 24.9441,C -1.727,E1 25.1592,E2 444.9245} C_DIS
LIN {X 115.6063,Y 13.2993,Z 125,A 2.8924,B 24.9436,C -1.7343,E1 25.1586,E2 443.0232} C_DIS
LIN {X 115.1683,Y 16.6735,Z 125,A 4.5937,B 24.9432,C -1.7409,E1 25.1579,E2 441.3163} C_DIS
LIN {X 114.5449,Y 20.5211,Z 125,A 6.4207,B 24.9431,C -1.7426,E1 25.1571,E2 439.4961} C_DIS
LIN {X 113.9481,Y 23.6118,Z 125,A 7.91,B 24.943,C -1.7446,E1 25.1563,E2 438.0108} C_DIS
LIN {X 113.3138,Y 26.49,Z 125,A 9.5003,B 24.9422,C -1.7558,E1 25.1553,E2 436.4032} C_DIS
LIN {X 112.1929,Y 30.8987,Z 125,A 11.5138,B 24.9425,C -1.7519,E1 25.1539,E2 434.4104} C_DIS
LIN {X 111.0469,Y 34.7901,Z 125,A 13.8671,B 24.9409,C -1.7751,E1 25.1519,E2 432.016} C_DIS
LIN {X 109.7156,Y 38.7842,Z 125,A 15.6433,B 24.9415,C -1.7671,E1 25.1503,E2 430.2685} C_DIS
LIN {X 108.5621,Y 41.9092,Z 125,A 17.2528,B 24.9412,C -1.7705,E1 25.1488,E2 428.66} C_DIS
LIN {X 107.3223,Y 44.9847,Z 125,A 18.9494,B 24.9407,C -1.7784,E1 25.1469,E2 426.9541} C_DIS
LIN {X 105.8006,Y 48.4602,Z 125,A 20.9188,B 24.94,C -1.7886,E1 25.1447,E2 424.9713} C_DIS
LIN {X 104.2807,Y 51.6448,Z 125,A 22.8619,B 24.939,C -1.8034,E1 25.1423,E2 423.0038} C_DIS
LIN {X 102.8107,Y 54.5134,Z 125,A 25.0454,B 24.9368,C -1.8364,E1 25.1393,E2 420.754} C_DIS
LIN {X 99.8807,Y 59.7145,Z 125,A 26.9499,B 24.9396,C -1.7949,E1 25.1368,E2 418.9571} C_DIS
LIN {X 98.3255,Y 62.2432,Z 125,A 28.6015,B 24.9387,C -1.8078,E1 25.1343,E2 417.2835} C_DIS
LIN {X 96.1947,Y 65.4852,Z 125,A 30.6661,B 24.9379,C -1.8201,E1 25.131,E2 415.2} C_DIS
LIN {X 93.1762,Y 69.7129,Z 125,A 32.9478,B 24.9384,C -1.8135,E1 25.1273,E2 412.9449} C_DIS
LIN {X 90.9855,Y 72.5502,Z 125,A 34.9136,B 24.9374,C -1.8272,E1 25.1239,E2 410.956} C_DIS
LIN {X 88.7623,Y 75.2527,Z 125,A 36.4055,B 24.9379,C -1.8204,E1 25.1212,E2 409.4869} C_DIS
LIN {X 86.6552,Y 77.6693,Z 125,A 37.9962,B 24.9376,C -1.8246,E1 25.1183,E2 407.8933} C_DIS
LIN {X 84.2484,Y 80.2764,Z 125,A 40.0107,B 24.9365,C -1.8411,E1 25.1144,E2 405.8489} C_DIS
LIN {X 80.5242,Y 84.0095,Z 125,A 42.3502,B 24.9369,C -1.8346,E1 25.1097,E2 403.5344} C_DIS
LIN {X 78.1534,Y 86.2217,Z 125,A 44.109,B 24.9362,C -1.8454,E1 25.1061,E2 401.7572} C_DIS
LIN {X 75.5671,Y 88.4945,Z 125,A 45.5823,B 24.9366,C -1.8385,E1 25.103,E2 400.3061} C_DIS
LIN {X 72.5849,Y 90.9581,Z 125,A 47.7145,B 24.9357,C -1.8526,E1 25.0983,E2 398.1485} C_DIS
LIN {X 68.6222,Y 93.9822,Z 125,A 49.8958,B 24.9362,C -1.8444,E1 25.0935,E2 395.9944} C_DIS
LIN {X 65.8685,Y 95.9345,Z 125,A 51.8299,B 24.9352,C -1.8598,E1 25.089,E2 394.0307} C_DIS
LIN {X 62.597,Y 98.0987,Z 125,A 53.5654,B 24.9356,C -1.8538,E1 25.085,E2 392.3149} C_DIS
LIN {X 58.8315,Y 100.4026,Z 125,A 55.6901,B 24.9356,C -1.8549,E1 25.0799,E2 390.1943} C_DIS
LIN {X 55.5464,Y 102.2558,Z 125,A 57.6786,B 24.9349,C -1.8635,E1 25.075,E2 388.1912} C_DIS
LIN {X 46.4083,Y 106.7142,Z 125,A 62.4445,B 24.9353,C -1.8585,E1 25.0631,E2 383.4494} C_DIS
LIN {X 43.3184,Y 108.007,Z 125,A 64.2393,B 24.9347,C -1.8669,E1 25.0584,E2 381.639} C_DIS
LIN {X 39.1592,Y 109.5839,Z 125,A 66.297,B 24.9349,C -1.8629,E1 25.053,E2 379.595} C_DIS
LIN {X 35.9353,Y 110.6811,Z 125,A 68.0735,B 24.9345,C -1.8689,E1 25.0483,E2 377.8079} C_DIS
LIN {X 31.5778,Y 112.0023,Z 125,A 70.2822,B 24.9345,C -1.869,E1 25.0424,E2 375.6027} C_DIS
LIN {X 27.2515,Y 113.1332,Z 125,A 72.3729,B 24.9348,C -1.8654,E1 25.0367,E2 373.5237} C_DIS
LIN {X 24.2667,Y 113.8115,Z 125,A 74.0687,B 24.9341,C -1.8746,E1 25.0321,E2 371.8083} C_DIS
LIN {X 20.661,Y 114.5197,Z 125,A 75.7318,B 24.9345,C -1.8688,E1 25.0275,E2 370.1608} C_DIS
LIN {X 17.809,Y 114.9977,Z 125,A 77.1629,B 24.9345,C -1.8696,E1 25.0236,E2 368.7293} C_DIS
LIN {X 14.5551,Y 115.4554,Z 125,A 78.8921,B 24.9341,C -1.8749,E1 25.0188,E2 366.989} C_DIS
LIN {X 10.3514,Y 115.9078,Z 125,A 80.8538,B 24.9345,C -1.8698,E1 25.0134,E2 365.0404} C_DIS
LIN {X 6.5955,Y 116.1816,Z 125,A 82.782,B 24.9342,C -1.8731,E1 25.008,E2 363.1052} C_DIS
LIN {X 3.0926,Y 116.3284,Z 125,A 84.5623,B 24.9341,C -1.8754,E1 25.003,E2 361.3201} C_DIS
LIN {X -0.6288,Y 116.3669,Z 125,A 86.317,B 24.9343,C -1.8716,E1 24.9981,E2 359.5743} C_DIS
LIN {X -4.5804,Y 116.2791,Z 125,A 88.2896,B 24.9343,C -1.8722,E1 24.9926,E2 357.6002} C_DIS
LIN {X -7.8619,Y 116.1027,Z 125,A 89.8228,B 24.9346,C -1.8678,E1 24.9884,E2 356.0767} C_DIS
LIN {X -11.0952,Y 115.8391,Z 125,A 91.5391,B 24.9343,C -1.8723,E1 24.9836,E2 354.349} C_DIS
LIN {X -14.9232,Y 115.4077,Z 125,A 93.3307,B 24.9347,C -1.8666,E1 24.9786,E2 352.5697} C_DIS
LIN {X -18.3974,Y 114.9068,Z 125,A 95.0421,B 24.9348,C -1.8646,E1 24.9739,E2 350.8615} C_DIS
LIN {X -21.7311,Y 114.3218,Z 125,A 96.6427,B 24.9351,C -1.8605,E1 24.9695,E2 349.269} C_DIS
LIN {X -26.496,Y 113.3121,Z 125,A 99.4739,B 24.9339,C -1.8771,E1 24.9617,E2 346.3949} C_DIS
LIN {X -29.6113,Y 112.54,Z 125,A 100.7185,B 24.9351,C -1.861,E1 24.9584,E2 345.1867} C_DIS
LIN {X -35.0668,Y 110.9611,Z 125,A 103.4884,B 24.9354,C -1.8567,E1 24.951,E2 342.4223} C_DIS
LIN {X -37.8269,Y 110.0509,Z 125,A 105.0662,B 24.9351,C -1.8612,E1 24.9468,E2 340.8309} C_DIS
LIN {X -41.2749,Y 108.8027,Z 125,A 107.0576,B 24.9347,C -1.8668,E1 24.9416,E2 338.822} C_DIS
LIN {X -45.2723,Y 107.2011,Z 125,A 108.9229,B 24.9356,C -1.8529,E1 24.9368,E2 336.9856} C_DIS
LIN {X -48.72,Y 105.6797,Z 125,A 110.9687,B 24.9353,C -1.8582,E1 24.9316,E2 334.9222} C_DIS
LIN {X -52.0303,Y 104.0896,Z 125,A 112.5867,B 24.936,C -1.8472,E1 24.9276,E2 333.3261} C_DIS
LIN {X -54.5915,Y 102.7696,Z 125,A 114.1401,B 24.9358,C -1.8505,E1 24.9237,E2 331.7606} C_DIS
LIN {X -58.0464,Y 100.8577,Z 125,A 115.9701,B 24.9364,C -1.8422,E1 24.9193,E2 329.9449} C_DIS
LIN {X -61.0236,Y 99.087,Z 125,A 117.6456,B 24.9367,C -1.8378,E1 24.9153,E2 328.2749} C_DIS
LIN {X -65.0711,Y 96.475,Z 125,A 120.8726,B 24.9345,C -1.8694,E1 24.9076,E2 324.962} C_DIS
LIN {X -69.4271,Y 93.3909,Z 125,A 123.3141,B 24.9354,C -1.8559,E1 24.9022,E2 322.5439} C_DIS
LIN {X -72.8862,Y 90.7166,Z 125,A 124.7148,B 24.9379,C -1.8196,E1 24.8993,E2 321.2245} C_DIS
LIN {X -74.7325,Y 89.2015,Z 125,A 126.1232,B 24.9375,C -1.8266,E1 24.8962,E2 319.7939} C_DIS
LIN {X -77.5184,Y 86.7903,Z 125,A 127.8492,B 24.938,C -1.8188,E1 24.8926,E2 318.0797} C_DIS
LIN {X -79.817,Y 84.6812,Z 125,A 129.4587,B 24.938,C -1.8182,E1 24.8893,E2 316.4649} C_DIS
LIN {X -82.8581,Y 81.7079,Z 125,A 131.5165,B 24.9385,C -1.8116,E1 24.8853,E2 314.4143} C_DIS
LIN {X -85.5424,Y 78.8937,Z 125,A 133.4805,B 24.9387,C -1.8089,E1 24.8815,E2 312.4483} C_DIS
LIN {X -87.6729,Y 76.5187,Z 125,A 135.0526,B 24.9389,C -1.8049,E1 24.8786,E2 310.8786} C_DIS
LIN {X -90.0943,Y 73.6539,Z 125,A 136.9376,B 24.9392,C -1.8016,E1 24.8752,E2 308.9928} C_DIS
LIN {X -92.6328,Y 70.4363,Z 125,A 139.5489,B 24.9379,C -1.8208,E1 24.8707,E2 306.3233} C_DIS
LIN {X -95.2624,Y 66.8354,Z 125,A 140.974,B 24.9404,C -1.7827,E1 24.8686,E2 304.9819} C_DIS
LIN {X -97.694,Y 63.2275,Z 125,A 143.3144,B 24.9403,C -1.7848,E1 24.8649,E2 302.6247} C_DIS
LIN {X -99.4984,Y 60.3466,Z 125,A 144.9677,B 24.9407,C -1.7792,E1 24.8625,E2 300.9764} C_DIS
LIN {X -102.3774,Y 55.3222,Z 125,A 147.7604,B 24.9414,C -1.7684,E1 24.8587,E2 298.1949} C_DIS
LIN {X -103.9044,Y 52.4015,Z 125,A 149.4017,B 24.9417,C -1.7643,E1 24.8566,E2 296.5546} C_DIS
LIN {X -105.1019,Y 49.9548,Z 125,A 150.882,B 24.9416,C -1.7659,E1 24.8548,E2 295.0623} C_DIS
LIN {X -106.6594,Y 46.534,Z 125,A 152.6616,B 24.9421,C -1.7574,E1 24.8528,E2 293.2933} C_DIS
LIN {X -107.9944,Y 43.3495,Z 125,A 154.5339,B 24.942,C -1.7592,E1 24.8508,E2 291.4063} C_DIS
LIN {X -109.2984,Y 39.9439,Z 125,A 156.1618,B 24.9428,C -1.7467,E1 24.8492,E2 289.7989} C_DIS
LIN {X -110.2997,Y 37.0893,Z 125,A 157.7137,B 24.943,C -1.7446,E1 24.8478,E2 288.2433} C_DIS
LIN {X -111.3563,Y 33.792,Z 125,A 159.5232,B 24.943,C -1.7434,E1 24.8463,E2 286.4262} C_DIS
LIN {X -112.3101,Y 30.4646,Z 125,A 161.1896,B 24.9435,C -1.7365,E1 24.845,E2 284.7666} C_DIS
LIN {X -113.2522,Y 26.7566,Z 125,A 163.2507,B 24.9435,C -1.7377,E1 24.8437,E2 282.6906} C_DIS
LIN {X -114.1618,Y 22.5622,Z 125,A 165.2416,B 24.9442,C -1.7258,E1 24.8426,E2 280.7162} C_DIS
LIN {X -114.882,Y 18.5501,Z 125,A 167.2242,B 24.9447,C -1.7183,E1 24.8416,E2 278.7398} C_DIS
LIN {X -115.3792,Y 15.1433,Z 125,A 168.8694,B 24.9452,C -1.7107,E1 24.841,E2 277.1028} C_DIS
LIN {X -115.8255,Y 11.2422,Z 125,A 170.7009,B 24.9458,C -1.7003,E1 24.8405,E2 275.2854} C_DIS
LIN {X -116.3247,Y 3.2131,Z 125,A 174.2834,B 24.9476,C -1.6719,E1 24.8399,E2 271.7489} C_DIS
LIN {X -116.3628,Y -1.3116,Z 125,A 177.1701,B 24.9464,C -1.6914,E1 24.8399,E2 268.7982} C_DIS
LIN {X -116.2538,Y -5.1693,Z 125,A 178.9884,B 24.947,C -1.6819,E1 24.84,E2 266.9916} C_DIS
LIN {X -116.0469,Y -8.6681,Z 125,A -178.4711,B 24.9452,C -1.71,E1 24.8406,E2 264.369} C_DIS
LIN {X -115.5355,Y -13.9045,Z 125,A -176.8667,B 24.9483,C -1.6609,E1 24.841,E2 262.872} C_DIS
LIN {X -114.873,Y -18.5997,Z 125,A -173.9953,B 24.9474,C -1.6755,E1 24.8422,E2 259.9486} C_DIS
LIN {X -113.7211,Y -24.6813,Z 125,A -171.5411,B 24.9495,C -1.6415,E1 24.8435,E2 257.5611} C_DIS
LIN {X -113.2033,Y -26.9639,Z 125,A -169.974,B 24.9487,C -1.6549,E1 24.8445,E2 255.9528} C_DIS
LIN {X -112.026,Y -31.494,Z 125,A -167.7638,B 24.9494,C -1.6439,E1 24.8461,E2 253.7559} C_DIS
LIN {X -111.0133,Y -34.8985,Z 125,A -166.0536,B 24.9498,C -1.6369,E1 24.8475,E2 252.0525} C_DIS
LIN {X -109.8618,Y -38.3673,Z 125,A -164.1924,B 24.95,C -1.6341,E1 24.8492,E2 250.1876} C_DIS
LIN {X -108.6141,Y -41.7729,Z 125,A -162.2858,B 24.95,C -1.6337,E1 24.8511,E2 248.2709} C_DIS
LIN {X -107.1632,Y -45.3621,Z 125,A -160.3109,B 24.9502,C -1.631,E1 24.8532,E2 246.2916} C_DIS
LIN {X -105.236,Y -49.673,Z 125,A -158.037,B 24.9507,C -1.6222,E1 24.8559,E2 244.0263} C_DIS
LIN {X -103.5988,Y -52.9993,Z 125,A -156.2807,B 24.9512,C -1.6142,E1 24.858,E2 242.2796} C_DIS
LIN {X -102.0365,Y -55.9506,Z 125,A -154.4767,B 24.951,C -1.6163,E1 24.8605,E2 240.461} C_DIS
LIN {X -100.0648,Y -59.4031,Z 125,A -152.6887,B 24.9518,C -1.604,E1 24.863,E2 238.6931} C_DIS
LIN {X -97.9107,Y -62.8899,Z 125,A -150.7098,B 24.9522,C -1.597,E1 24.8659,E2 236.7208} C_DIS
LIN {X -96.3037,Y -65.3242,Z 125,A -149.1192,B 24.952,C -1.5998,E1 24.8684,E2 235.1157} C_DIS
LIN {X -94.171,Y -68.3644,Z 125,A -147.3085,B 24.9524,C -1.5944,E1 24.8713,E2 233.309} C_DIS
LIN {X -91.7298,Y -71.6084,Z 125,A -145.236,B 24.9524,C -1.5926,E1 24.8749,E2 231.231} C_DIS
LIN {X -89.42,Y -74.4696,Z 125,A -143.5464,B 24.953,C -1.5832,E1 24.8778,E2 229.5558} C_DIS
LIN {X -87.4796,Y -76.7399,Z 125,A -142.028,B 24.9531,C -1.5818,E1 24.8806,E2 228.0338} C_DIS
LIN {X -84.8555,Y -79.6316,Z 125,A -140.1604,B 24.9535,C -1.5752,E1 24.8841,E2 226.1738} C_DIS
LIN {X -82.5377,Y -82.0323,Z 125,A -138.3779,B 24.9534,C -1.5775,E1 24.8876,E2 224.3781} C_DIS
LIN {X -79.7125,Y -84.7795,Z 125,A -136.5328,B 24.9539,C -1.5694,E1 24.8913,E2 222.5446} C_DIS
LIN {X -77.3757,Y -86.918,Z 125,A -134.9145,B 24.9539,C -1.5688,E1 24.8947,E2 220.9214} C_DIS
LIN {X -73.8658,Y -89.9218,Z 125,A -132.7479,B 24.9544,C -1.5598,E1 24.8993,E2 218.7679} C_DIS
LIN {X -71.3239,Y -91.9493,Z 125,A -131.0145,B 24.9543,C -1.5625,E1 24.9031,E2 217.0216} C_DIS
LIN {X -68.2153,Y -94.2801,Z 125,A -128.9856,B 24.9542,C -1.5641,E1 24.9077,E2 214.9817} C_DIS
LIN {X -64.9245,Y -96.5743,Z 125,A -127.1018,B 24.9546,C -1.5569,E1 24.9121,E2 213.1086} C_DIS
LIN {X -61.3196,Y -98.9025,Z 125,A -125.101,B 24.9551,C -1.5488,E1 24.9167,E2 211.1208} C_DIS
LIN {X -58.6539,Y -100.5076,Z 125,A -123.3794,B 24.9547,C -1.5547,E1 24.9209,E2 209.3798} C_DIS
LIN {X -55.4947,Y -102.2838,Z 125,A -121.7464,B 24.9552,C -1.5458,E1 24.9249,E2 207.7635} C_DIS
LIN {X -49.86,Y -105.1474,Z 125,A -118.6703,B 24.9556,C -1.5402,E1 24.9326,E2 204.6924} C_DIS
LIN {X -46.802,Y -106.5426,Z 125,A -116.9295,B 24.9554,C -1.5421,E1 24.937,E2 202.9428} C_DIS
LIN {X -43.2755,Y -108.0242,Z 125,A -115.1667,B 24.9559,C -1.5349,E1 24.9415,E2 201.1933} C_DIS
LIN {X -40.5042,Y -109.094,Z 125,A -113.6729,B 24.9559,C -1.5349,E1 24.9454,E2 199.6964} C_DIS
LIN {X -37.7029,Y -110.0929,Z 125,A -112.1727,B 24.9559,C -1.5352,E1 24.9494,E2 198.1925} C_DIS
LIN {X -34.2632,Y -111.2103,Z 125,A -110.3779,B 24.9559,C -1.5345,E1 24.9542,E2 196.3963} C_DIS
LIN {X -30.1621,Y -112.3919,Z 125,A -108.244,B 24.9559,C -1.5345,E1 24.9599,E2 194.2589} C_DIS
LIN {X -26.4305,Y -113.3275,Z 125,A -106.2969,B 24.9559,C -1.5358,E1 24.9652,E2 192.306} C_DIS
LIN {X -22.676,Y -114.1399,Z 125,A -104.3244,B 24.9556,C -1.5386,E1 24.9706,E2 190.3246} C_DIS
LIN {X -18.9797,Y -114.8105,Z 125,A -102.5782,B 24.9559,C -1.5334,E1 24.9754,E2 188.589} C_DIS
LIN {X -14.9317,Y -115.4066,Z 125,A -100.7123,B 24.9564,C -1.5263,E1 24.9805,E2 186.7384} C_DIS
LIN {X -12.2393,Y -115.7232,Z 125,A -99.2731,B 24.9561,C -1.5308,E1 24.9846,E2 185.2877} C_DIS
LIN {X -9.1367,Y -116.0094,Z 125,A -97.7053,B 24.9561,C -1.5323,E1 24.9889,E2 183.7157} C_DIS
LIN {X -6.0677,Y -116.2108,Z 125,A -96.2499,B 24.9561,C -1.5297,E1 24.993,E2 182.266} C_DIS
LIN {X -3.0765,Y -116.3289,Z 125,A -94.8152,B 24.9563,C -1.5281,E1 24.997,E2 180.8348} C_DIS
LIN {X -0.4289,Y -116.3681,Z 125,A -93.4669,B 24.9561,C -1.5304,E1 25.0008,E2 179.4811} C_DIS
LIN {X -0.4289,Y -116.3681,Z 125,A -93.4669,B 24.9561,C -1.5304,E1 25.0008,E2 179.4811} C_DIS
Enddeposition()
LIN {X 0.83,Y -115.5,Z 125,A -93.421,B 24.9567,C -1.52,E1 25.0008,E2 179.4598} C_DIS
Startdeposition()
$VEL.CP = VEL_PRINT
LIN {X -1.8466,Y -115.4903,Z 125,A -94.674,B 24.9565,C -1.523,E1 24.9973,E2 180.7057} C_DIS
LIN {X -4.7314,Y -115.408,Z 125,A -96.2846,B 24.957,C -1.5149,E1 24.9928,E2 182.3357} C_DIS
LIN {X -7.4688,Y -115.2634,Z 125,A -97.4756,B 24.9566,C -1.5223,E1 24.9895,E2 183.5097} C_DIS
LIN {X -10.3761,Y -115.038,Z 125,A -98.882,B 24.9565,C -1.5241,E1 24.9856,E2 184.9123} C_DIS
LIN {X -12.7291,Y -114.8034,Z 125,A -100.2651,B 24.957,C -1.5149,E1 24.9817,E2 186.318} C_DIS
LIN {X -16.0088,Y -114.3902,Z 125,A -101.9446,B 24.957,C -1.5136,E1 24.977,E2 188.0019} C_DIS
LIN {X -18.9144,Y -113.9456,Z 125,A -103.3362,B 24.9569,C -1.5169,E1 24.9732,E2 189.387} C_DIS
LIN {X -22.9932,Y -113.1933,Z 125,A -105.423,B 24.9569,C -1.5164,E1 24.9675,E2 191.4772} C_DIS
LIN {X -27.1374,Y -112.2718,Z 125,A -107.5953,B 24.957,C -1.5146,E1 24.9616,E2 193.6566} C_DIS
LIN {X -30.0935,Y -111.5156,Z 125,A -108.9956,B 24.9567,C -1.5204,E1 24.9578,E2 195.0451} C_DIS
LIN {X -33.5354,Y -110.5315,Z 125,A -110.9849,B 24.9571,C -1.5124,E1 24.9524,E2 197.0567} C_DIS
LIN {X -36.6819,Y -109.5255,Z 125,A -112.5263,B 24.9568,C -1.5179,E1 24.9484,E2 198.5878} C_DIS
LIN {X -40.2443,Y -108.2693,Z 125,A -114.345,B 24.9566,C -1.5219,E1 24.9436,E2 200.4007} C_DIS
LIN {X -43.2003,Y -107.1224,Z 125,A -115.7752,B 24.9562,C -1.5296,E1 24.9399,E2 201.8158} C_DIS
LIN {X -45.9413,Y -105.9754,Z 125,A -117.4154,B 24.9565,C -1.524,E1 24.9357,E2 203.4729} C_DIS
LIN {X -48.3528,Y -104.8977,Z 125,A -118.6184,B 24.9561,C -1.5301,E1 24.9326,E2 204.6646} C_DIS
LIN {X -51.1171,Y -103.5781,Z 125,A -120.0291,B 24.9558,C -1.5365,E1 24.9291,E2 206.0635} C_DIS
LIN {X -53.2139,Y -102.5188,Z 125,A -121.3991,B 24.9562,C -1.5293,E1 24.9256,E2 207.4544} C_DIS
LIN {X -55.9539,Y -101.0479,Z 125,A -122.8178,B 24.9558,C -1.5367,E1 24.9222,E2 208.8596} C_DIS
LIN {X -58.5663,Y -99.556,Z 125,A -124.2379,B 24.9555,C -1.5419,E1 24.9188,E2 210.2716} C_DIS
LIN {X -60.987,Y -98.0918,Z 125,A -125.6497,B 24.9554,C -1.5436,E1 24.9154,E2 211.6836} C_DIS
LIN {X -63.3816,Y -96.5618,Z 125,A -127.321,B 24.9559,C -1.5348,E1 24.9114,E2 213.3813} C_DIS
LIN {X -65.7442,Y -94.9689,Z 125,A -128.6875,B 24.9556,C -1.5391,E1 24.9083,E2 214.7421} C_DIS
LIN {X -68.0472,Y -93.3326,Z 125,A -130.0942,B 24.9555,C -1.5413,E1 24.9051,E2 216.1485} C_DIS
LIN {X -70.5023,Y -91.4919,Z 125,A -131.6679,B 24.9555,C -1.5418,E1 24.9016,E2 217.7265} C_DIS
LIN {X -73.2683,Y -89.2949,Z 125,A -133.4752,B 24.9555,C -1.5428,E1 24.8976,E2 219.5384} C_DIS
LIN {X -75.8068,Y -87.1477,Z 125,A -135.0985,B 24.9552,C -1.5471,E1 24.8942,E2 221.1577} C_DIS
LIN {X -78.2695,Y -84.9428,Z 125,A -136.7395,B 24.955,C -1.5504,E1 24.8908,E2 222.7975} C_DIS
LIN {X -81.0034,Y -82.3398,Z 125,A -138.6286,B 24.9548,C -1.5536,E1 24.887,E2 224.6867} C_DIS
LIN {X -83.2109,Y -80.1081,Z 125,A -140.163,B 24.9545,C -1.558,E1 24.884,E2 226.2174} C_DIS
LIN {X -85.5866,Y -77.5679,Z 125,A -141.9535,B 24.9545,C -1.5591,E1 24.8806,E2 228.0131} C_DIS
LIN {X -87.6089,Y -75.2746,Z 125,A -143.392,B 24.9541,C -1.5658,E1 24.878,E2 229.442} C_DIS
LIN {X -89.6336,Y -72.8505,Z 125,A -145.0066,B 24.954,C -1.5676,E1 24.8751,E2 231.0598} C_DIS
LIN {X -91.9298,Y -69.9339,Z 125,A -146.8137,B 24.9536,C -1.5735,E1 24.8721,E2 232.8616} C_DIS
LIN {X -93.6142,Y -67.6625,Z 125,A -148.225,B 24.9534,C -1.5766,E1 24.8697,E2 234.2723} C_DIS
LIN {X -95.2425,Y -65.3506,Z 125,A -149.6361,B 24.9532,C -1.5799,E1 24.8675,E2 235.6826} C_DIS
LIN {X -97.0643,Y -62.6093,Z 125,A -151.2733,B 24.953,C -1.5839,E1 24.865,E2 237.3182} C_DIS
LIN {X -98.5786,Y -60.1969,Z 125,A -152.7318,B 24.9529,C -1.5858,E1 24.8628,E2 238.7798} C_DIS
LIN {X -100.0377,Y -57.7395,Z 125,A -154.1235,B 24.9526,C -1.5907,E1 24.8609,E2 240.167} C_DIS
LIN {X -101.4196,Y -55.2762,Z 125,A -155.5329,B 24.9524,C -1.5942,E1 24.859,E2 241.5755} C_DIS
LIN {X -103.1732,Y -51.934,Z 125,A -157.5746,B 24.9524,C -1.5926,E1 24.8563,E2 243.6321} C_DIS
LIN {X -104.6083,Y -48.9746,Z 125,A -159.058,B 24.9518,C -1.6032,E1 24.8546,E2 245.0981} C_DIS
LIN {X -106.345,Y -45.0794,Z 125,A -161.1877,B 24.9515,C -1.6088,E1 24.8522,E2 247.2263} C_DIS
LIN {X -107.5023,Y -42.2446,Z 125,A -162.6578,B 24.9511,C -1.6152,E1 24.8507,E2 248.6892} C_DIS
LIN {X -108.9105,Y -38.4695,Z 125,A -164.5177,B 24.9504,C -1.6268,E1 24.8489,E2 250.5321} C_DIS
LIN {X -109.6771,Y -36.2324,Z 125,A -166.0674,B 24.9511,C -1.6151,E1 24.8475,E2 252.1185} C_DIS
LIN {X -110.937,Y -32.1688,Z 125,A -168.1976,B 24.9508,C -1.6208,E1 24.8458,E2 254.2475} C_DIS
LIN {X -111.697,Y -29.421,Z 125,A -169.6209,B 24.9505,C -1.6248,E1 24.8447,E2 255.6695} C_DIS
LIN {X -112.7002,Y -25.3083,Z 125,A -171.6385,B 24.9499,C -1.6346,E1 24.8435,E2 257.6754} C_DIS
LIN {X -113.3969,Y -21.966,Z 125,A -173.0762,B 24.949,C -1.6503,E1 24.8427,E2 259.0843} C_DIS
LIN {X -113.893,Y -19.2294,Z 125,A -174.6605,B 24.9492,C -1.6464,E1 24.8419,E2 260.6872} C_DIS
LIN {X -114.517,Y -15.0748,Z 125,A -176.8053,B 24.9489,C -1.6506,E1 24.841,E2 262.8348} C_DIS
LIN {X -114.9474,Y -11.353,Z 125,A -178.7805,B 24.9489,C -1.6519,E1 24.8404,E2 264.8188} C_DIS
LIN {X -115.2895,Y -7.083,Z 125,A 179.2243,B 24.9481,C -1.664,E1 24.84,E2 266.7971} C_DIS
LIN {X -115.4427,Y -3.7931,Z 125,A 177.5157,B 24.948,C -1.6663,E1 24.8398,E2 268.5105} C_DIS
LIN {X -115.5048,Y -0.421,Z 125,A 175.8326,B 24.9477,C -1.6713,E1 24.8398,E2 270.1918} C_DIS
LIN {X -115.472,Y 2.8387,Z 125,A 174.1502,B 24.9475,C -1.674,E1 24.8398,E2 271.8779} C_DIS
LIN {X -115.3329,Y 6.2989,Z 125,A 172.4546,B 24.9471,C -1.6805,E1 24.8401,E2 273.5682} C_DIS
LIN {X -115.056,Y 10.1807,Z 125,A 170.6905,B 24.9463,C -1.6934,E1 24.8405,E2 275.3121} C_DIS
LIN {X -114.7988,Y 12.768,Z 125,A 169.2959,B 24.9463,C -1.6934,E1 24.8409,E2 276.7151} C_DIS
LIN {X -114.3877,Y 16.0267,Z 125,A 167.8606,B 24.9454,C -1.7065,E1 24.8414,E2 278.1277} C_DIS
LIN {X -114.0383,Y 18.3603,Z 125,A 166.3176,B 24.9461,C -1.6954,E1 24.8421,E2 279.7064} C_DIS
LIN {X -113.5554,Y 21.1427,Z 125,A 164.9056,B 24.9459,C -1.6995,E1 24.8428,E2 281.117} C_DIS
LIN {X -112.6989,Y 25.3141,Z 125,A 162.7786,B 24.9455,C -1.7057,E1 24.844,E2 283.2417} C_DIS
LIN {X -111.69,Y 29.4479,Z 125,A 160.6531,B 24.9451,C -1.7119,E1 24.8455,E2 285.3649} C_DIS
LIN {X -110.5332,Y 33.53,Z 125,A 158.533,B 24.9447,C -1.718,E1 24.8471,E2 287.4827} C_DIS
LIN {X -109.2271,Y 37.5668,Z 125,A 156.4159,B 24.9443,C -1.7241,E1 24.849,E2 289.5972} C_DIS
LIN {X -108.2746,Y 40.2299,Z 125,A 155.1589,B 24.9436,C -1.7343,E1 24.8502,E2 290.837} C_DIS
LIN {X -107.2482,Y 42.8913,Z 125,A 153.5633,B 24.9438,C -1.7315,E1 24.8518,E2 292.4483} C_DIS
LIN {X -105.5922,Y 46.82,Z 125,A 151.607,B 24.943,C -1.7443,E1 24.854,E2 294.3848} C_DIS
LIN {X -104.414,Y 49.3918,Z 125,A 150.036,B 24.9431,C -1.7419,E1 24.8559,E2 295.9702} C_DIS
LIN {X -103.1731,Y 51.9341,Z 125,A 148.6862,B 24.9427,C -1.7482,E1 24.8575,E2 297.3121} C_DIS
LIN {X -101.8406,Y 54.5,Z 125,A 147.3425,B 24.9422,C -1.7561,E1 24.8593,E2 298.6442} C_DIS
LIN {X -100.4835,Y 56.9637,Z 125,A 145.7812,B 24.9424,C -1.7536,E1 24.8614,E2 300.2197} C_DIS
LIN {X -99.0644,Y 59.3975,Z 125,A 144.3727,B 24.9421,C -1.7572,E1 24.8634,E2 301.627} C_DIS
LIN {X -97.5854,Y 61.7975,Z 125,A 142.9638,B 24.9419,C -1.7608,E1 24.8655,E2 303.0345} C_DIS
LIN {X -95.7889,Y 64.5438,Z 125,A 141.4843,B 24.9412,C -1.7713,E1 24.8678,E2 304.4961} C_DIS
LIN {X -94.1866,Y 66.8604,Z 125,A 140.0795,B 24.941,C -1.7749,E1 24.87,E2 305.8994} C_DIS
LIN {X -92.5314,Y 69.133,Z 125,A 138.5942,B 24.941,C -1.7751,E1 24.8725,E2 307.3914} C_DIS
LIN {X -90.4661,Y 71.8143,Z 125,A 136.9281,B 24.9406,C -1.7801,E1 24.8753,E2 309.0534} C_DIS
LIN {X -88.227,Y 74.5491,Z 125,A 135.144,B 24.9404,C -1.7835,E1 24.8785,E2 310.8378} C_DIS
LIN {X -86.059,Y 77.0402,Z 125,A 133.5291,B 24.94,C -1.7887,E1 24.8815,E2 312.4475} C_DIS
LIN {X -83.6547,Y 79.6476,Z 125,A 131.6403,B 24.94,C -1.7878,E1 24.8851,E2 314.3467} C_DIS
LIN {X -81.1651,Y 82.1801,Z 125,A 130.0346,B 24.9394,C -1.7985,E1 24.8883,E2 315.9337} C_DIS
LIN {X -78.9598,Y 84.3015,Z 125,A 128.4544,B 24.9394,C -1.7996,E1 24.8915,E2 317.5179} C_DIS
LIN {X -76.3449,Y 86.6778,Z 125,A 126.748,B 24.9389,C -1.8055,E1 24.895,E2 319.2169} C_DIS
LIN {X -73.9029,Y 88.7677,Z 125,A 125.1885,B 24.9386,C -1.8105,E1 24.8983,E2 320.7705} C_DIS
LIN {X -71.5247,Y 90.695,Z 125,A 123.5543,B 24.9386,C -1.8091,E1 24.9019,E2 322.4142} C_DIS
LIN {X -68.7551,Y 92.8143,Z 125,A 121.8893,B 24.9382,C -1.8154,E1 24.9056,E2 324.0701} C_DIS
LIN {X -66.4869,Y 94.4527,Z 125,A 120.4936,B 24.9381,C -1.8179,E1 24.9088,E2 325.4647} C_DIS
LIN {X -64.1748,Y 96.0387,Z 125,A 118.9242,B 24.9384,C -1.8134,E1 24.9124,E2 327.0502} C_DIS
LIN {X -61.7752,Y 97.5994,Z 125,A 117.5099,B 24.9382,C -1.8163,E1 24.9158,E2 328.462} C_DIS
LIN {X -59.3692,Y 99.0814,Z 125,A 116.1013,B 24.938,C -1.8186,E1 24.9191,E2 329.8694} C_DIS
LIN {X -56.5217,Y 100.7308,Z 125,A 114.619,B 24.9374,C -1.8278,E1 24.9227,E2 331.3344} C_DIS
LIN {X -54.0396,Y 102.0839,Z 125,A 113.2114,B 24.9372,C -1.8299,E1 24.9261,E2 332.7407} C_DIS
LIN {X -50.2565,Y 103.9985,Z 125,A 111.0929,B 24.937,C -1.8327,E1 24.9314,E2 334.8583} C_DIS
LIN {X -46.8056,Y 105.5987,Z 125,A 109.0455,B 24.9373,C -1.8289,E1 24.9367,E2 336.9198} C_DIS
LIN {X -43.7383,Y 106.9034,Z 125,A 107.5499,B 24.9367,C -1.8379,E1 24.9405,E2 338.3975} C_DIS
LIN {X -40.2273,Y 108.2755,Z 125,A 105.5182,B 24.937,C -1.8336,E1 24.9458,E2 340.4435} C_DIS
LIN {X -37.1904,Y 109.354,Z 125,A 104.2512,B 24.9359,C -1.8495,E1 24.949,E2 341.6751} C_DIS
LIN {X -34.4,Y 110.2634,Z 125,A 102.8162,B 24.9357,C -1.8521,E1 24.9529,E2 343.1065} C_DIS
LIN {X -32.1505,Y 110.9421,Z 125,A 101.2893,B 24.9367,C -1.8382,E1 24.957,E2 344.6691} C_DIS
LIN {X -29.1704,Y 111.7614,Z 125,A 99.9461,B 24.936,C -1.8478,E1 24.9606,E2 345.9916} C_DIS
LIN {X -26.142,Y 112.5076,Z 125,A 98.5635,B 24.9354,C -1.8562,E1 24.9643,E2 347.356} C_DIS
LIN {X -23.4984,Y 113.0895,Z 125,A 97.0061,B 24.936,C -1.8483,E1 24.9686,E2 348.9341} C_DIS
LIN {X -21.1265,Y 113.5583,Z 125,A 95.6529,B 24.9363,C -1.8428,E1 24.9724,E2 350.302} C_DIS
LIN {X -16.9415,Y 114.2577,Z 125,A 93.5439,B 24.9363,C -1.844,E1 24.9782,E2 352.4099} C_DIS
LIN {X -13.6768,Y 114.6924,Z 125,A 92.0188,B 24.9359,C -1.8497,E1 24.9824,E2 353.9227} C_DIS
LIN {X -10.4791,Y 115.0285,Z 125,A 90.4361,B 24.9358,C -1.851,E1 24.9868,E2 355.5031} C_DIS
LIN {X -7.0744,Y 115.29,Z 125,A 88.7732,B 24.9356,C -1.853,E1 24.9914,E2 357.1619} C_DIS
LIN {X -3.7845,Y 115.443,Z 125,A 87.1378,B 24.9356,C -1.8535,E1 24.9959,E2 358.7964} C_DIS
LIN {X -0.8309,Y 115.5018,Z 125,A 85.6322,B 24.9356,C -1.8521,E1 25.0002,E2 360.3054} C_DIS
LIN {X 2.3764,Y 115.4806,Z 125,A 84.0249,B 24.9357,C -1.8517,E1 25.0046,E2 361.9135} C_DIS
LIN {X 6.137,Y 115.3418,Z 125,A 82.1872,B 24.9357,C -1.853,E1 25.0098,E2 363.7475} C_DIS
LIN {X 10.3724,Y 115.0383,Z 125,A 80.3133,B 24.9349,C -1.863,E1 25.0149,E2 365.5968} C_DIS
LIN {X 13.1441,Y 114.7548,Z 125,A 78.6717,B 24.9357,C -1.8515,E1 25.0195,E2 367.2645} C_DIS
LIN {X 16.9585,Y 114.2551,Z 125,A 76.8184,B 24.9357,C -1.8534,E1 25.0247,E2 369.1118} C_DIS
LIN {X 20.2087,Y 113.7234,Z 125,A 75.394,B 24.935,C -1.862,E1 25.0285,E2 370.5144} C_DIS
LIN {X 22.988,Y 113.1943,Z 125,A 73.7827,B 24.9357,C -1.8523,E1 25.033,E2 372.1468} C_DIS
LIN {X 25.6747,Y 112.6156,Z 125,A 72.3851,B 24.9358,C -1.8501,E1 25.0368,E2 373.5477} C_DIS
LIN {X 29.4504,Y 111.6893,Z 125,A 70.3413,B 24.9363,C -1.8438,E1 25.0424,E2 375.6033} C_DIS
LIN {X 33.5393,Y 110.5303,Z 125,A 68.2346,B 24.9363,C -1.8424,E1 25.048,E2 377.7098} C_DIS
LIN {X 37.5746,Y 109.2245,Z 125,A 66.1335,B 24.9365,C -1.8407,E1 25.0536,E2 379.8108} C_DIS
LIN {X 40.2556,Y 108.265,Z 125,A 64.881,B 24.9361,C -1.8464,E1 25.0568,E2 381.0471} C_DIS
LIN {X 42.895,Y 107.2467,Z 125,A 63.3533,B 24.9366,C -1.8395,E1 25.0608,E2 382.5878} C_DIS
LIN {X 46.0557,Y 105.9256,Z 125,A 61.9821,B 24.9357,C -1.8523,E1 25.0643,E2 383.9256} C_DIS
LIN {X 48.1663,Y 104.9845,Z 125,A 60.6503,B 24.9364,C -1.8426,E1 25.0677,E2 385.2769} C_DIS
LIN {X 51.1027,Y 103.5852,Z 125,A 59.2423,B 24.9359,C -1.8499,E1 25.0712,E2 386.6641} C_DIS
LIN {X 53.1922,Y 102.5302,Z 125,A 57.8695,B 24.9366,C -1.8388,E1 25.0747,E2 388.0592} C_DIS
LIN {X 55.7004,Y 101.1894,Z 125,A 56.4683,B 24.9367,C -1.8373,E1 25.0781,E2 389.4599} C_DIS
LIN {X 58.5608,Y 99.5592,Z 125,A 55.0436,B 24.9362,C -1.8443,E1 25.0815,E2 390.8638} C_DIS
LIN {X 60.9928,Y 98.0881,Z 125,A 53.5142,B 24.9368,C -1.8368,E1 25.0852,E2 392.4063} C_DIS
LIN {X 63.4009,Y 96.549,Z 125,A 52.0227,B 24.9371,C -1.8312,E1 25.0887,E2 393.906} C_DIS
LIN {X 65.7395,Y 94.9722,Z 125,A 50.6284,B 24.9373,C -1.8291,E1 25.0919,E2 395.3006} C_DIS
LIN {X 68.04,Y 93.3379,Z 125,A 49.2337,B 24.9374,C -1.8269,E1 25.0951,E2 396.6957} C_DIS
LIN {X 70.4941,Y 91.4983,Z 125,A 47.668,B 24.9378,C -1.8221,E1 25.0986,E2 398.2669} C_DIS
LIN {X 73.2799,Y 89.2854,Z 125,A 45.815,B 24.9383,C -1.8147,E1 25.1026,E2 400.1304} C_DIS
LIN {X 75.8189,Y 87.1372,Z 125,A 44.2599,B 24.9382,C -1.8158,E1 25.1059,E2 401.6769} C_DIS
LIN {X 78.2626,Y 84.9492,Z 125,A 42.64,B 24.9384,C -1.8128,E1 25.1093,E2 403.2974} C_DIS
LIN {X 81.0064,Y 82.3369,Z 125,A 40.7621,B 24.9387,C -1.8089,E1 25.113,E2 405.1767} C_DIS
LIN {X 83.1696,Y 80.1509,Z 125,A 39.2637,B 24.9388,C -1.8068,E1 25.116,E2 406.6736} C_DIS
LIN {X 85.5869,Y 77.5676,Z 125,A 37.4715,B 24.9392,C -1.8011,E1 25.1194,E2 408.4714} C_DIS
LIN {X 87.7641,Y 75.0924,Z 125,A 36.0045,B 24.9389,C -1.805,E1 25.122,E2 409.9224} C_DIS
LIN {X 89.4477,Y 73.0799,Z 125,A 34.5282,B 24.9397,C -1.7939,E1 25.1247,E2 411.4183} C_DIS
LIN {X 91.4954,Y 70.4977,Z 125,A 32.9665,B 24.9397,C -1.7932,E1 25.1273,E2 412.9741} C_DIS
LIN {X 93.6084,Y 67.6706,Z 125,A 31.1779,B 24.9401,C -1.7871,E1 25.1303,E2 414.7687} C_DIS
LIN {X 95.2489,Y 65.3412,Z 125,A 29.8659,B 24.9401,C -1.7881,E1 25.1324,E2 416.0718} C_DIS
LIN {X 97.0725,Y 62.5966,Z 125,A 28.2188,B 24.9404,C -1.7833,E1 25.1349,E2 417.722} C_DIS
LIN {X 99.1133,Y 59.3151,Z 125,A 26.192,B 24.9411,C -1.7731,E1 25.1379,E2 419.7626} C_DIS
LIN {X 100.7432,Y 56.4995,Z 125,A 24.7337,B 24.9409,C -1.7759,E1 25.1399,E2 421.2067} C_DIS
LIN {X 102.1477,Y 53.9185,Z 125,A 23.3237,B 24.941,C -1.774,E1 25.1418,E2 422.6137} C_DIS
LIN {X 104.0067,Y 50.2395,Z 125,A 21.2481,B 24.9415,C -1.7668,E1 25.1443,E2 424.6953} C_DIS
LIN {X 105.5964,Y 46.8108,Z 125,A 19.2277,B 24.9423,C -1.7546,E1 25.1467,E2 426.7335} C_DIS
LIN {X 106.908,Y 43.7271,Z 125,A 17.743,B 24.9421,C -1.758,E1 25.1483,E2 428.2019} C_DIS
LIN {X 108.2707,Y 40.2406,Z 125,A 15.7322,B 24.9429,C -1.7453,E1 25.1503,E2 430.2316} C_DIS
LIN {X 109.2233,Y 37.5781,Z 125,A 14.4842,B 24.9427,C -1.7483,E1 25.1514,E2 431.4655} C_DIS
LIN {X 110.2539,Y 34.4306,Z 125,A 12.8533,B 24.943,C -1.7439,E1 25.1528,E2 433.0976} C_DIS
LIN {X 111.4399,Y 30.3737,Z 125,A 10.9785,B 24.9427,C -1.7478,E1 25.1543,E2 434.9523} C_DIS
LIN {X 112.0446,Y 28.0687,Z 125,A 9.4447,B 24.9441,C -1.7276,E1 25.1554,E2 436.5249} C_DIS
LIN {X 112.7022,Y 25.2993,Z 125,A 8.2028,B 24.9438,C -1.7312,E1 25.1561,E2 437.7513} C_DIS
LIN {X 113.3758,Y 22.0755,Z 125,A 6.7873,B 24.9435,C -1.7363,E1 25.1569,E2 439.1465} C_DIS
LIN {X 113.8825,Y 19.2921,Z 125,A 5.1851,B 24.9444,C -1.7225,E1 25.1577,E2 440.7718} C_DIS
LIN {X 114.3369,Y 16.3841,Z 125,A 3.6933,B 24.9448,C -1.7163,E1 25.1583,E2 442.2693} C_DIS
LIN {X 114.6931,Y 13.6708,Z 125,A 2.3874,B 24.9449,C -1.7144,E1 25.1588,E2 443.5721} C_DIS
LIN {X 115.1181,Y 9.4464,Z 125,A 0.2957,B 24.9453,C -1.7082,E1 25.1593,E2 445.6659} C_DIS
LIN {X 115.3923,Y 5.0967,Z 125,A -1.8213,B 24.9456,C -1.7033,E1 25.1597,E2 447.7818} C_DIS
LIN {X 115.4808,Y 2.3638,Z 125,A -3.1732,B 24.9459,C -1.6991,E1 25.1597,E2 449.1357} C_DIS
LIN {X 115.5056,Y -0.2824,Z 125,A -4.3983,B 24.9459,C -1.699,E1 25.1597,E2 450.3538} C_DIS
LIN {X 115.4722,Y -2.8325,Z 125,A -5.914,B 24.9469,C -1.683,E1 25.1597,E2 451.8981} C_DIS
LIN {X 115.289,Y -7.0916,Z 125,A -7.8577,B 24.9469,C -1.6841,E1 25.1594,E2 453.8276} C_DIS
LIN {X 115.037,Y -10.3865,Z 125,A -9.276,B 24.9465,C -1.6892,E1 25.1591,E2 455.2256} C_DIS
LIN {X 114.803,Y -12.7326,Z 125,A -10.6476,B 24.9474,C -1.6758,E1 25.1587,E2 456.6207} C_DIS
LIN {X 114.3914,Y -16.0003,Z 125,A -12.0656,B 24.9471,C -1.6807,E1 25.1582,E2 458.0187} C_DIS
LIN {X 114.0417,Y -18.339,Z 125,A -13.6174,B 24.9484,C -1.659,E1 25.1575,E2 459.6126} C_DIS
LIN {X 113.506,Y -21.3993,Z 125,A -15.0684,B 24.9484,C -1.6582,E1 25.1568,E2 461.0569} C_DIS
LIN {X 112.7941,Y -24.878,Z 125,A -16.7682,B 24.9486,C -1.6554,E1 25.1558,E2 462.7534} C_DIS
LIN {X 111.9208,Y -28.5505,Z 125,A -18.3702,B 24.9482,C -1.6621,E1 25.1548,E2 464.3302} C_DIS
LIN {X 111.1918,Y -31.2693,Z 125,A -19.9588,B 24.9491,C -1.6486,E1 25.1536,E2 465.9418} C_DIS
LIN {X 109.9739,Y -35.3149,Z 125,A -22.051,B 24.9495,C -1.6421,E1 25.1519,E2 468.0374} C_DIS
LIN {X 108.5928,Y -39.3574,Z 125,A -23.9409,B 24.9492,C -1.6462,E1 25.1502,E2 469.907} C_DIS
LIN {X 107.7661,Y -41.573,Z 125,A -25.3126,B 24.95,C -1.6331,E1 25.1488,E2 471.3018} C_DIS
LIN {X 106.6538,Y -44.3465,Z 125,A -26.8983,B 24.9506,C -1.6236,E1 25.1471,E2 472.9011} C_DIS
LIN {X 105.5822,Y -46.8422,Z 125,A -28.1202,B 24.9505,C -1.6254,E1 25.1457,E2 474.1123} C_DIS
LIN {X 104.4083,Y -49.4037,Z 125,A -29.6645,B 24.9512,C -1.6142,E1 25.1439,E2 475.6745} C_DIS
LIN {X 103.1713,Y -51.9377,Z 125,A -30.9002,B 24.951,C -1.6176,E1 25.1424,E2 476.8956} C_DIS
LIN {X 101.8725,Y -54.4409,Z 125,A -32.2925,B 24.9512,C -1.6137,E1 25.1406,E2 478.2897} C_DIS
LIN {X 100.5134,Y -56.911,Z 125,A -33.8392,B 24.9519,C -1.6027,E1 25.1384,E2 479.8544} C_DIS
LIN {X 99.075,Y -59.38,Z 125,A -35.2454,B 24.9521,C -1.599,E1 25.1364,E2 481.262} C_DIS
LIN {X 97.5849,Y -61.7983,Z 125,A -36.6541,B 24.9523,C -1.595,E1 25.1343,E2 482.6732} C_DIS
LIN {X 95.7671,Y -64.5759,Z 125,A -38.1255,B 24.9521,C -1.5985,E1 25.1321,E2 484.1289} C_DIS
LIN {X 94.1624,Y -66.8943,Z 125,A -39.5159,B 24.9523,C -1.595,E1 25.1298,E2 485.5208} C_DIS
LIN {X 92.5011,Y -69.1734,Z 125,A -40.9745,B 24.9527,C -1.5883,E1 25.1274,E2 486.9882} C_DIS
LIN {X 90.474,Y -71.8043,Z 125,A -42.6394,B 24.953,C -1.583,E1 25.1245,E2 488.6576} C_DIS
LIN {X 88.1933,Y -74.5886,Z 125,A -44.388,B 24.9532,C -1.58,E1 25.1214,E2 490.4053} C_DIS
LIN {X 86.0548,Y -77.0449,Z 125,A -45.9738,B 24.9534,C -1.5772,E1 25.1185,E2 491.9907} C_DIS
LIN {X 83.6514,Y -79.651,Z 125,A -47.8354,B 24.9539,C -1.5679,E1 25.1149,E2 493.866} C_DIS
LIN {X 81.4216,Y -81.9268,Z 125,A -49.3568,B 24.954,C -1.5668,E1 25.1119,E2 495.3837} C_DIS
LIN {X 78.9355,Y -84.3243,Z 125,A -51.0028,B 24.954,C -1.5657,E1 25.1086,E2 497.0253} C_DIS
LIN {X 76.3315,Y -86.6895,Z 125,A -52.6896,B 24.9542,C -1.5643,E1 25.1051,E2 498.7088} C_DIS
LIN {X 74.1851,Y -88.5332,Z 125,A -54.0866,B 24.9543,C -1.5614,E1 25.1021,E2 500.1072} C_DIS
LIN {X 71.7827,Y -90.4911,Z 125,A -55.6731,B 24.9547,C -1.5557,E1 25.0987,E2 501.7011} C_DIS
LIN {X 69.1731,Y -92.5013,Z 125,A -57.2936,B 24.9548,C -1.5528,E1 25.095,E2 503.3226} C_DIS
LIN {X 66.5193,Y -94.4299,Z 125,A -58.8659,B 24.9548,C -1.5519,E1 25.0915,E2 504.8916} C_DIS
LIN {X 64.1709,Y -96.0414,Z 125,A -60.4448,B 24.9555,C -1.5415,E1 25.0878,E2 506.4898} C_DIS
LIN {X 61.5027,Y -97.7696,Z 125,A -61.8989,B 24.9553,C -1.544,E1 25.0844,E2 507.9332} C_DIS
LIN {X 59.3296,Y -99.1048,Z 125,A -63.2468,B 24.9557,C -1.5378,E1 25.0811,E2 509.2915} C_DIS
LIN {X 56.4996,Y -100.7432,Z 125,A -64.7138,B 24.9555,C -1.542,E1 25.0776,E2 510.7443} C_DIS
LIN {X 54.0289,Y -102.0895,Z 125,A -66.1046,B 24.9555,C -1.5398,E1 25.0742,E2 512.1363} C_DIS
LIN {X 50.2285,Y -104.012,Z 125,A -68.2118,B 24.9558,C -1.5365,E1 25.0689,E2 514.2456} C_DIS
LIN {X 46.8003,Y -105.601,Z 125,A -70.2358,B 24.9563,C -1.5268,E1 25.0637,E2 516.2876} C_DIS
LIN {X 43.7691,Y -106.8909,Z 125,A -71.7577,B 24.9562,C -1.5295,E1 25.0598,E2 517.7995} C_DIS
LIN {X 40.1501,Y -108.3037,Z 125,A -73.7694,B 24.9565,C -1.523,E1 25.0546,E2 519.8223} C_DIS
LIN {X 37.5253,Y -109.2411,Z 125,A -75.0022,B 24.9563,C -1.5279,E1 25.0513,E2 521.0409} C_DIS
LIN {X 34.4258,Y -110.2554,Z 125,A -76.6728,B 24.9565,C -1.5236,E1 25.0469,E2 522.7186} C_DIS
LIN {X 30.3896,Y -111.4356,Z 125,A -78.5108,B 24.956,C -1.5324,E1 25.042,E2 524.5325} C_DIS
LIN {X 28.0588,Y -112.047,Z 125,A -80.0533,B 24.957,C -1.5155,E1 25.0377,E2 526.1127} C_DIS
LIN {X 25.3033,Y -112.7013,Z 125,A -81.298,B 24.9566,C -1.5214,E1 25.0344,E2 527.342} C_DIS
LIN {X 22.0795,Y -113.375,Z 125,A -82.9829,B 24.9568,C -1.5177,E1 25.0298,E2 529.0334} C_DIS
LIN {X 19.0192,Y -113.9281,Z 125,A -84.402,B 24.9566,C -1.522,E1 25.0259,E2 530.4409} C_DIS
LIN {X 15.0759,Y -114.5169,Z 125,A -86.444,B 24.9568,C -1.5177,E1 25.0202,E2 532.4912} C_DIS
LIN {X 11.3217,Y -114.9507,Z 125,A -88.4808,B 24.9573,C -1.5094,E1 25.0145,E2 534.5463} C_DIS
LIN {X 7.0667,Y -115.2904,Z 125,A -90.431,B 24.957,C -1.5158,E1 25.0091,E2 536.4803} C_DIS
LIN {X 3.7777,Y -115.4432,Z 125,A -92.0636,B 24.957,C -1.5153,E1 25.0046,E2 538.1137} C_DIS
LIN {X 0.83,Y -115.5,Z 125,A -93.4201,B 24.9567,C -1.5196,E1 25.0008,E2 539.4598} C_DIS
Enddeposition()
LIN {X 0.8591,Y -121.2409,Z 126,A -92.8173,B 24.9604,C -1.4543,E1 25.0021,E2 539.0118} C_DIS
Startdeposition()
$VEL.CP = VEL_PRINT
LIN {X 4.5821,Y -121.1602,Z 126,A -90.9011,B 24.9599,C -1.4622,E1 25.0075,E2 537.0773} C_DIS
LIN {X 7.435,Y -121.0193,Z 126,A -89.5912,B 24.96,C -1.4609,E1 25.0111,E2 535.7711} C_DIS
LIN {X 10.4027,Y -120.8004,Z 126,A -88.1866,B 24.96,C -1.4615,E1 25.015,E2 534.3657} C_DIS
LIN {X 13.3642,Y -120.5088,Z 126,A -86.7819,B 24.96,C -1.4622,E1 25.0189,E2 532.9602} C_DIS
LIN {X 16.3176,Y -120.1445,Z 126,A -85.2207,B 24.9595,C -1.4706,E1 25.0233,E2 531.3805} C_DIS
LIN {X 19.2612,Y -119.7078,Z 126,A -83.9738,B 24.9599,C -1.464,E1 25.0267,E2 530.1504} C_DIS
LIN {X 22.1931,Y -119.1991,Z 126,A -82.4764,B 24.9595,C -1.4695,E1 25.0308,E2 528.6417} C_DIS
LIN {X 25.1117,Y -118.6186,Z 126,A -81.1601,B 24.9597,C -1.4664,E1 25.0344,E2 527.3343} C_DIS
LIN {X 28.0152,Y -117.9666,Z 126,A -79.7629,B 24.9597,C -1.4673,E1 25.0382,E2 525.9369} C_DIS
LIN {X 30.9018,Y -117.2435,Z 126,A -78.3595,B 24.9596,C -1.4687,E1 25.042,E2 524.5325} C_DIS
LIN {X 33.7698,Y -116.4498,Z 126,A -76.9567,B 24.9596,C -1.4701,E1 25.0458,E2 523.1287} C_DIS
LIN {X 36.6175,Y -115.586,Z 126,A -75.5542,B 24.9594,C -1.4716,E1 25.0495,E2 521.7251} C_DIS
LIN {X 39.4431,Y -114.6525,Z 126,A -74.1515,B 24.9594,C -1.4732,E1 25.0532,E2 520.3213} C_DIS
LIN {X 42.2449,Y -113.65,Z 126,A -72.7494,B 24.9593,C -1.4749,E1 25.0569,E2 518.9182} C_DIS
LIN {X 45.0213,Y -112.5791,Z 126,A -71.3474,B 24.9592,C -1.4766,E1 25.0606,E2 517.5151} C_DIS
LIN {X 47.7706,Y -111.4403,Z 126,A -69.9457,B 24.959,C -1.4785,E1 25.0642,E2 516.1123} C_DIS
LIN {X 50.4911,Y -110.2344,Z 126,A -68.3924,B 24.9585,C -1.4879,E1 25.0682,E2 514.5408} C_DIS
LIN {X 53.7003,Y -108.7047,Z 126,A -66.8698,B 24.9588,C -1.483,E1 25.072,E2 513.0337} C_DIS
LIN {X 57.1557,Y -106.9308,Z 126,A -65.0406,B 24.9586,C -1.4858,E1 25.0765,E2 511.203} C_DIS
LIN {X 59.926,Y -105.402,Z 126,A -63.437,B 24.9582,C -1.4938,E1 25.0804,E2 509.5852} C_DIS
LIN {X 62.3337,Y -103.9975,Z 126,A -62.2394,B 24.9584,C -1.4904,E1 25.0833,E2 508.3993} C_DIS
LIN {X 64.8671,Y -102.4364,Z 126,A -60.67,B 24.9578,C -1.5011,E1 25.087,E2 506.8096} C_DIS
LIN {X 68.5936,Y -99.9794,Z 126,A -58.7385,B 24.958,C -1.4966,E1 25.0915,E2 504.8952} C_DIS
LIN {X 71.0265,Y -98.2659,Z 126,A -57.3385,B 24.9579,C -1.4992,E1 25.0947,E2 503.4939} C_DIS
LIN {X 73.4893,Y -96.4373,Z 126,A -55.9343,B 24.9579,C -1.5001,E1 25.0978,E2 502.0927} C_DIS
LIN {X 75.7627,Y -94.6625,Z 126,A -54.5389,B 24.9576,C -1.5047,E1 25.1009,E2 500.6916} C_DIS
LIN {X 78.063,Y -92.7746,Z 126,A -53.1394,B 24.9574,C -1.5076,E1 25.1039,E2 499.2907} C_DIS
LIN {X 80.3163,Y -90.8309,Z 126,A -51.7402,B 24.9573,C -1.5105,E1 25.1068,E2 497.8901} C_DIS
LIN {X 82.5212,Y -88.8325,Z 126,A -50.3412,B 24.9571,C -1.5135,E1 25.1097,E2 496.4897} C_DIS
LIN {X 84.6764,Y -86.7806,Z 126,A -48.9418,B 24.9569,C -1.5166,E1 25.1125,E2 495.0888} C_DIS
LIN {X 86.7806,Y -84.6764,Z 126,A -47.5431,B 24.9567,C -1.5197,E1 25.1153,E2 493.6888} C_DIS
LIN {X 88.8325,Y -82.5212,Z 126,A -46.1447,B 24.9565,C -1.5229,E1 25.1179,E2 492.2889} C_DIS
LIN {X 90.8309,Y -80.3163,Z 126,A -44.746,B 24.9564,C -1.5262,E1 25.1205,E2 490.8887} C_DIS
LIN {X 92.7746,Y -78.063,Z 126,A -43.1996,B 24.9557,C -1.5369,E1 25.1234,E2 489.3241} C_DIS
LIN {X 94.6625,Y -75.7627,Z 126,A -41.9494,B 24.956,C -1.5329,E1 25.1255,E2 488.0892} C_DIS
LIN {X 96.4932,Y -73.4167,Z 126,A -40.5515,B 24.9558,C -1.5363,E1 25.1279,E2 486.6899} C_DIS
LIN {X 98.2659,Y -71.0265,Z 126,A -39.1533,B 24.9556,C -1.5398,E1 25.1302,E2 485.2901} C_DIS
LIN {X 99.9794,Y -68.5936,Z 126,A -37.7556,B 24.9554,C -1.5434,E1 25.1325,E2 483.8909} C_DIS
LIN {X 101.6327,Y -66.1193,Z 126,A -36.3578,B 24.9552,C -1.5469,E1 25.1346,E2 482.4916} C_DIS
LIN {X 103.2836,Y -63.5083,Z 126,A -34.9548,B 24.9551,C -1.5483,E1 25.1367,E2 481.0924} C_DIS
LIN {X 104.7546,Y -61.0528,Z 126,A -33.5625,B 24.9547,C -1.5543,E1 25.1387,E2 479.6933} C_DIS
LIN {X 106.2213,Y -58.4636,Z 126,A -32.1655,B 24.9545,C -1.558,E1 25.1406,E2 478.2948} C_DIS
LIN {X 107.6241,Y -55.8392,Z 126,A -30.7678,B 24.9543,C -1.5618,E1 25.1424,E2 476.8955} C_DIS
LIN {X 109.1996,Y -52.6868,Z 126,A -29.1052,B 24.954,C -1.5667,E1 25.1444,E2 475.2302} C_DIS
LIN {X 110.8457,Y -49.1345,Z 126,A -27.2749,B 24.9537,C -1.5714,E1 25.1466,E2 473.3988} C_DIS
LIN {X 112.1408,Y -46.0981,Z 126,A -25.6538,B 24.9533,C -1.5793,E1 25.1483,E2 471.7679} C_DIS
LIN {X 113.65,Y -42.2449,Z 126,A -23.7827,B 24.9532,C -1.5812,E1 25.1502,E2 469.9028} C_DIS
LIN {X 114.6525,Y -39.4431,Z 126,A -22.3857,B 24.9529,C -1.5852,E1 25.1515,E2 468.5043} C_DIS
LIN {X 115.586,Y -36.6175,Z 126,A -20.9891,B 24.9527,C -1.5892,E1 25.1527,E2 467.1062} C_DIS
LIN {X 116.4498,Y -33.7698,Z 126,A -19.5922,B 24.9524,C -1.5932,E1 25.1538,E2 465.7078} C_DIS
LIN {X 117.2435,Y -30.9018,Z 126,A -18.1957,B 24.9522,C -1.5972,E1 25.1548,E2 464.3098} C_DIS
LIN {X 117.9666,Y -28.0152,Z 126,A -16.7993,B 24.952,C -1.6013,E1 25.1557,E2 462.9119} C_DIS
LIN {X 118.6186,Y -25.1117,Z 126,A -15.4026,B 24.9517,C -1.6054,E1 25.1565,E2 461.5137} C_DIS
LIN {X 119.1991,Y -22.1931,Z 126,A -14.006,B 24.9515,C -1.6095,E1 25.1573,E2 460.1157} C_DIS
LIN {X 119.7187,Y -19.1913,Z 126,A -12.6059,B 24.9513,C -1.6122,E1 25.1579,E2 458.7173} C_DIS
LIN {X 120.1445,Y -16.3176,Z 126,A -11.213,B 24.951,C -1.6177,E1 25.1585,E2 457.3196} C_DIS
Enddeposition()
END
